LIN {X 0,Y 380.592,Z 511.818,A -85,B 0,C 180,E1 -13079.719,E2 -13079.719} C_VEL
LIN {X 0,Y 375.84,Z 486.306,A -85,B 0,C 180,E1 -13080.73,E2 -13080.73} C_VEL
LIN {X 0,Y 368.954,Z 471.038,A -85,B 0,C 180,E1 -13081.761,E2 -13081.761} C_VEL
LIN {X 0,Y 368.004,Z 468.713,A -85,B 0,C 180,E1 -13081.936,E2 -13081.936} C_VEL
LIN {X 0,Y 364.375,Z 454.654,A -85,B 0,C 180,E1 -13085.353,E2 -13085.353} C_VEL
LIN {X 0,Y 361.868,Z 446.029,A -85,B 0,C 180,E1 -13087.61,E2 -13087.61} C_VEL
LIN {X 0,Y 361.87,Z 446.036,A -85,B 0,C 180,E1 -13091.323,E2 -13091.323} C_VEL
LIN {X 0,Y 361.898,Z 446.033,A -85,B 0,C 180,E1 -13094.354,E2 -13094.354} C_VEL
LIN {X 0,Y 361.831,Z 446.035,A -85,B 0,C 180,E1 -13097.567,E2 -13097.567} C_VEL
LIN {X 0,Y 361.865,Z 446.035,A -85,B 0,C 180,E1 -13100.973,E2 -13100.973} C_VEL
LIN {X 0,Y 361.868,Z 446.032,A -85,B 0,C 180,E1 -13104.655,E2 -13104.655} C_VEL
LIN {X 0,Y 361.831,Z 446.041,A -85,B 0,C 180,E1 -13108.37,E2 -13108.37} C_VEL
LIN {X 0,Y 361.901,Z 446.029,A -85,B 0,C 180,E1 -13112.221,E2 -13112.221} C_VEL
LIN {X 0,Y 361.921,Z 446.028,A -85,B 0,C 180,E1 -13114.71,E2 -13114.71} C_VEL
LIN {X 0,Y 361.885,Z 446.032,A -85,B 0,C 180,E1 -13118.347,E2 -13118.347} C_VEL
LIN {X 0,Y 361.96,Z 446.023,A -85,B 0,C 180,E1 -13122.061,E2 -13122.061} C_VEL
LIN {X 0,Y 361.991,Z 446.016,A -85,B 0,C 180,E1 -13126.101,E2 -13126.101} C_VEL
LIN {X 0,Y 362.029,Z 446.01,A -85,B 0,C 180,E1 -13129.938,E2 -13129.938} C_VEL
LIN {X 0,Y 362.144,Z 446.001,A -85,B 0,C 180,E1 -13132.193,E2 -13132.193} C_VEL
LIN {X 0,Y 362.112,Z 445.999,A -85,B 0,C 180,E1 -13134.431,E2 -13134.431} C_VEL
LIN {X 0,Y 362.276,Z 445.977,A -85,B 0,C 180,E1 -13137.777,E2 -13137.777} C_VEL
LIN {X 0,Y 362.421,Z 445.967,A -85,B 0,C 180,E1 -13140,E2 -13140} C_VEL
LIN {X 0,Y 362.276,Z 445.979,A -85,B 0,C 180,E1 -13142.224,E2 -13142.224} C_VEL
LIN {X 0,Y 362.165,Z 445.997,A -85,B 0,C 180,E1 -13146.687,E2 -13146.687} C_VEL
LIN {X 0,Y 362.067,Z 446.01,A -85,B 0,C 180,E1 -13148.934,E2 -13148.934} C_VEL
LIN {X 0,Y 361.954,Z 446.024,A -85,B 0,C 180,E1 -13152.333,E2 -13152.333} C_VEL
LIN {X 0,Y 361.957,Z 446.022,A -85,B 0,C 180,E1 -13154.621,E2 -13154.621} C_VEL
LIN {X 0,Y 361.954,Z 446.026,A -85,B 0,C 180,E1 -13158.1,E2 -13158.1} C_VEL
LIN {X 0,Y 361.886,Z 446.03,A -85,B 0,C 180,E1 -13161.654,E2 -13161.654} C_VEL
LIN {X 0,Y 361.923,Z 446.03,A -85,B 0,C 180,E1 -13165.291,E2 -13165.291} C_VEL
LIN {X 0,Y 361.917,Z 446.03,A -85,B 0,C 180,E1 -13167.779,E2 -13167.779} C_VEL
LIN {X 0,Y 361.855,Z 446.037,A -85,B 0,C 180,E1 -13171.628,E2 -13171.628} C_VEL
LIN {X 0,Y 361.898,Z 446.125,A -85,B 0,C 180,E1 -13173.963,E2 -13173.963} C_VEL
LIN {X 0,Y 363.631,Z 452.4,A -85,B 0,C 180,E1 -13175.693,E2 -13175.693} C_VEL
LIN {X 0,Y 374.505,Z 473.576,A -85,B 0,C 180,E1 -13177.307,E2 -13177.307} C_VEL
LIN {X 0,Y 381.161,Z 488.749,A -85,B 0,C 180,E1 -13178.277,E2 -13178.277} C_VEL
LIN {X 0,Y 377.634,Z 617.32,A -85,B 0,C 180,E1 -13180.831,E2 -13180.831} C_VEL
LIN {X 0,Y 376.702,Z 633.034,A -85,B 0,C 180,E1 -13181.362,E2 -13181.362} C_VEL
LIN {X 0,Y 375.589,Z 647.26,A -85,B 0,C 180,E1 -13182.05,E2 -13182.05} C_VEL
LIN {X 0,Y 374.132,Z 661.968,A -85,B 0,C 180,E1 -13182.995,E2 -13182.995} C_VEL
LIN {X 0,Y 372.388,Z 676.407,A -85,B 0,C 180,E1 -13184.181,E2 -13184.181} C_VEL
LIN {X 0,Y 370.685,Z 688.967,A -85,B 0,C 180,E1 -13185.454,E2 -13185.454} C_VEL
LIN {X 0,Y 368.931,Z 700.675,A -85,B 0,C 180,E1 -13186.891,E2 -13186.891} C_VEL
LIN {X 0,Y 367.053,Z 712.573,A -85,B 0,C 180,E1 -13188.658,E2 -13188.658} C_VEL
LIN {X 0,Y 365.247,Z 723.245,A -85,B 0,C 180,E1 -13190.583,E2 -13190.583} C_VEL
LIN {X 0,Y 364.044,Z 731.254,A -85,B 0,C 180,E1 -13192.328,E2 -13192.328} C_VEL
LIN {X 0,Y 362.703,Z 739.466,A -85,B 0,C 180,E1 -13194.472,E2 -13194.472} C_VEL
LIN {X 0,Y 361.751,Z 746.21,A -85,B 0,C 180,E1 -13196.657,E2 -13196.657} C_VEL
LIN {X 0,Y 361.075,Z 751.703,A -85,B 0,C 180,E1 -13198.918,E2 -13198.918} C_VEL
LIN {X 0,Y 360.532,Z 756.05,A -85,B 0,C 180,E1 -13201.308,E2 -13201.308} C_VEL
LIN {X 0,Y 360.22,Z 759.126,A -85,B 0,C 180,E1 -13203.829,E2 -13203.829} C_VEL
LIN {X 0,Y 360.067,Z 760.813,A -85,B 0,C 180,E1 -13206.546,E2 -13206.546} C_VEL
LIN {X 0,Y 360.056,Z 760.99,A -85,B 0,C 180,E1 -13208.232,E2 -13208.232} C_VEL
LIN {X 0,Y 360.152,Z 760.166,A -85,B 0,C 180,E1 -13210.627,E2 -13210.627} C_VEL
LIN {X 0,Y 360.35,Z 758.07,A -85,B 0,C 180,E1 -13212.99,E2 -13212.99} C_VEL
LIN {X 0,Y 360.698,Z 754.681,A -85,B 0,C 180,E1 -13215.328,E2 -13215.328} C_VEL
LIN {X 0,Y 361.143,Z 749.972,A -85,B 0,C 180,E1 -13217.64,E2 -13217.64} C_VEL
LIN {X 0,Y 361.874,Z 743.855,A -85,B 0,C 180,E1 -13219.934,E2 -13219.934} C_VEL
LIN {X 0,Y 362.924,Z 736.176,A -85,B 0,C 180,E1 -13222.21,E2 -13222.21} C_VEL
LIN {X 0,Y 364.092,Z 727.96,A -85,B 0,C 180,E1 -13224.184,E2 -13224.184} C_VEL
LIN {X 0,Y 365.644,Z 718.092,A -85,B 0,C 180,E1 -13226.144,E2 -13226.144} C_VEL
LIN {X 0,Y 367.185,Z 708.015,A -85,B 0,C 180,E1 -13227.807,E2 -13227.807} C_VEL
LIN {X 0,Y 368.887,Z 696.077,A -85,B 0,C 180,E1 -13229.455,E2 -13229.455} C_VEL
LIN {X 0,Y 370.57,Z 684.121,A -85,B 0,C 180,E1 -13230.816,E2 -13230.816} C_VEL
LIN {X 0,Y 372.187,Z 671.209,A -85,B 0,C 180,E1 -13232.03,E2 -13232.03} C_VEL
LIN {X 0,Y 373.735,Z 656.677,A -85,B 0,C 180,E1 -13233.128,E2 -13233.128} C_VEL
LIN {X 0,Y 374.985,Z 642.461,A -85,B 0,C 180,E1 -13233.963,E2 -13233.963} C_VEL
LIN {X 0,Y 376.031,Z 627.288,A -85,B 0,C 180,E1 -13234.624,E2 -13234.624} C_VEL
LIN {X 0,Y 376.736,Z 611.413,A -85,B 0,C 180,E1 -13235.084,E2 -13235.084} C_VEL
LIN {X 0,Y 377.665,Z 575.869,A -85,B 0,C 180,E1 -13235.78,E2 -13235.78} C_VEL
LIN {X 0,Y 377.269,Z 570.066,A -85,B 0,C 180,E1 -13235.934,E2 -13235.934} C_VEL
LIN {X 0,Y 372.626,Z 551.43,A -85,B 0,C 180,E1 -13236.7,E2 -13236.7} C_VEL
LIN {X 0,Y 372.167,Z 545.629,A -85,B 0,C 180,E1 -13236.864,E2 -13236.864} C_VEL
LIN {X 0,Y 373.609,Z 489.608,A -85,B 0,C 180,E1 -13237.975,E2 -13237.975} C_VEL
LIN {X 0,Y 364.5,Z 468.659,A -85,B 0,C 180,E1 -13239.245,E2 -13239.245} C_VEL
LIN {X 0,Y 356.131,Z 451.447,A -85,B 0,C 180,E1 -13240.457,E2 -13240.457} C_VEL
LIN {X 0,Y 354.915,Z 446.893,A -85,B 0,C 180,E1 -13241.711,E2 -13241.711} C_VEL
LIN {X 0,Y 354.924,Z 446.901,A -85,B 0,C 180,E1 -13244.917,E2 -13244.917} C_VEL
LIN {X 0,Y 354.913,Z 446.898,A -85,B 0,C 180,E1 -13248.472,E2 -13248.472} C_VEL
LIN {X 0,Y 354.842,Z 446.912,A -85,B 0,C 180,E1 -13252.106,E2 -13252.106} C_VEL
LIN {X 0,Y 354.903,Z 446.904,A -85,B 0,C 180,E1 -13255.827,E2 -13255.827} C_VEL
LIN {X 0,Y 354.858,Z 446.907,A -85,B 0,C 180,E1 -13259.679,E2 -13259.679} C_VEL
LIN {X 0,Y 354.809,Z 446.907,A -85,B 0,C 180,E1 -13263.702,E2 -13263.702} C_VEL
LIN {X 0,Y 354.802,Z 446.91,A -85,B 0,C 180,E1 -13266.459,E2 -13266.459} C_VEL
LIN {X 0,Y 354.827,Z 446.904,A -85,B 0,C 180,E1 -13269.424,E2 -13269.424} C_VEL
LIN {X 0,Y 354.793,Z 446.908,A -85,B 0,C 180,E1 -13272.867,E2 -13272.867} C_VEL
LIN {X 0,Y 354.778,Z 446.916,A -85,B 0,C 180,E1 -13276.105,E2 -13276.105} C_VEL
LIN {X 0,Y 354.826,Z 446.901,A -85,B 0,C 180,E1 -13279.184,E2 -13279.184} C_VEL
LIN {X 0,Y 354.811,Z 446.908,A -85,B 0,C 180,E1 -13282.402,E2 -13282.402} C_VEL
LIN {X 0,Y 354.814,Z 446.902,A -85,B 0,C 180,E1 -13284.941,E2 -13284.941} C_VEL
LIN {X 0,Y 354.797,Z 446.909,A -85,B 0,C 180,E1 -13288.404,E2 -13288.404} C_VEL
LIN {X 0,Y 354.848,Z 446.901,A -85,B 0,C 180,E1 -13291.618,E2 -13291.618} C_VEL
LIN {X 0,Y 354.9,Z 446.899,A -85,B 0,C 180,E1 -13294.172,E2 -13294.172} C_VEL
LIN {X 0,Y 354.828,Z 446.902,A -85,B 0,C 180,E1 -13297.893,E2 -13297.893} C_VEL
LIN {X 0,Y 354.924,Z 446.89,A -85,B 0,C 180,E1 -13301.891,E2 -13301.891} C_VEL
LIN {X 0,Y 354.944,Z 446.897,A -85,B 0,C 180,E1 -13305.981,E2 -13305.981} C_VEL
LIN {X 0,Y 354.979,Z 446.878,A -85,B 0,C 180,E1 -13309.736,E2 -13309.736} C_VEL
LIN {X 0,Y 355.115,Z 446.871,A -85,B 0,C 180,E1 -13312.037,E2 -13312.037} C_VEL
LIN {X 0,Y 355.093,Z 446.875,A -85,B 0,C 180,E1 -13314.32,E2 -13314.32} C_VEL
LIN {X 0,Y 355.244,Z 446.846,A -85,B 0,C 180,E1 -13317.732,E2 -13317.732} C_VEL
LIN {X 0,Y 355.398,Z 446.841,A -85,B 0,C 180,E1 -13320,E2 -13320} C_VEL
LIN {X 0,Y 355.246,Z 446.851,A -85,B 0,C 180,E1 -13322.267,E2 -13322.267} C_VEL
LIN {X 0,Y 355.138,Z 446.865,A -85,B 0,C 180,E1 -13326.819,E2 -13326.819} C_VEL
LIN {X 0,Y 355.015,Z 446.886,A -85,B 0,C 180,E1 -13329.112,E2 -13329.112} C_VEL
LIN {X 0,Y 354.921,Z 446.884,A -85,B 0,C 180,E1 -13332.581,E2 -13332.581} C_VEL
LIN {X 0,Y 354.889,Z 446.901,A -85,B 0,C 180,E1 -13336.096,E2 -13336.096} C_VEL
LIN {X 0,Y 354.901,Z 446.884,A -85,B 0,C 180,E1 -13338.472,E2 -13338.472} C_VEL
LIN {X 0,Y 354.835,Z 446.909,A -85,B 0,C 180,E1 -13342.106,E2 -13342.106} C_VEL
LIN {X 0,Y 354.899,Z 446.901,A -85,B 0,C 180,E1 -13345.827,E2 -13345.827} C_VEL
LIN {X 0,Y 354.854,Z 446.91,A -85,B 0,C 180,E1 -13349.678,E2 -13349.678} C_VEL
LIN {X 0,Y 354.806,Z 446.913,A -85,B 0,C 180,E1 -13353.702,E2 -13353.702} C_VEL
LIN {X 0,Y 354.801,Z 446.913,A -85,B 0,C 180,E1 -13356.459,E2 -13356.459} C_VEL
LIN {X 0,Y 354.824,Z 446.913,A -85,B 0,C 180,E1 -13359.423,E2 -13359.423} C_VEL
LIN {X 0,Y 354.791,Z 446.914,A -85,B 0,C 180,E1 -13362.867,E2 -13362.867} C_VEL
LIN {X 0,Y 354.851,Z 446.907,A -85,B 0,C 180,E1 -13366.116,E2 -13366.116} C_VEL
LIN {X 0,Y 354.856,Z 446.909,A -85,B 0,C 180,E1 -13369.188,E2 -13369.188} C_VEL
LIN {X 0,Y 354.832,Z 446.935,A -85,B 0,C 180,E1 -13372.597,E2 -13372.597} C_VEL
LIN {X 0,Y 358.374,Z 460.009,A -85,B 0,C 180,E1 -13375.824,E2 -13375.824} C_VEL
LIN {X 0,Y 360.621,Z 469.402,A -85,B 0,C 180,E1 -13378.014,E2 -13378.014} C_VEL
LIN {X 0,Y 368.425,Z 487.379,A -85,B 0,C 180,E1 -13379.138,E2 -13379.138} C_VEL
LIN {X 0,Y 373.23,Z 513.749,A -85,B 0,C 180,E1 -13380.135,E2 -13380.135} C_VEL
LIN {X 0,Y 369.957,Z 635.975,A -85,B 0,C 180,E1 -13382.569,E2 -13382.569} C_VEL
LIN {X 0,Y 368.945,Z 652.02,A -85,B 0,C 180,E1 -13383.101,E2 -13383.101} C_VEL
LIN {X 0,Y 367.762,Z 666.067,A -85,B 0,C 180,E1 -13383.773,E2 -13383.773} C_VEL
LIN {X 0,Y 366.127,Z 681.117,A -85,B 0,C 180,E1 -13384.724,E2 -13384.724} C_VEL
LIN {X 0,Y 364.458,Z 694.507,A -85,B 0,C 180,E1 -13385.809,E2 -13385.809} C_VEL
LIN {X 0,Y 362.564,Z 708.251,A -85,B 0,C 180,E1 -13387.189,E2 -13387.189} C_VEL
LIN {X 0,Y 360.698,Z 720.702,A -85,B 0,C 180,E1 -13388.721,E2 -13388.721} C_VEL
LIN {X 0,Y 359.084,Z 731.85,A -85,B 0,C 180,E1 -13390.384,E2 -13390.384} C_VEL
LIN {X 0,Y 357.371,Z 742.327,A -85,B 0,C 180,E1 -13392.252,E2 -13392.252} C_VEL
LIN {X 0,Y 355.992,Z 751.579,A -85,B 0,C 180,E1 -13394.249,E2 -13394.249} C_VEL
LIN {X 0,Y 354.917,Z 759.263,A -85,B 0,C 180,E1 -13396.253,E2 -13396.253} C_VEL
LIN {X 0,Y 354.138,Z 766.441,A -85,B 0,C 180,E1 -13398.553,E2 -13398.553} C_VEL
LIN {X 0,Y 353.593,Z 772.091,A -85,B 0,C 180,E1 -13400.85,E2 -13400.85} C_VEL
LIN {X 0,Y 353.305,Z 776.376,A -85,B 0,C 180,E1 -13403.145,E2 -13403.145} C_VEL
LIN {X 0,Y 353.226,Z 779.396,A -85,B 0,C 180,E1 -13405.435,E2 -13405.435} C_VEL
LIN {X 0,Y 353.161,Z 781.216,A -85,B 0,C 180,E1 -13407.718,E2 -13407.718} C_VEL
LIN {X 0,Y 353.26,Z 781.847,A -85,B 0,C 180,E1 -13409.999,E2 -13409.999} C_VEL
LIN {X 0,Y 353.163,Z 781.288,A -85,B 0,C 180,E1 -13412.28,E2 -13412.28} C_VEL
LIN {X 0,Y 353.23,Z 779.582,A -85,B 0,C 180,E1 -13414.564,E2 -13414.564} C_VEL
LIN {X 0,Y 353.307,Z 776.695,A -85,B 0,C 180,E1 -13416.854,E2 -13416.854} C_VEL
LIN {X 0,Y 353.595,Z 772.565,A -85,B 0,C 180,E1 -13419.148,E2 -13419.148} C_VEL
LIN {X 0,Y 354.147,Z 767.089,A -85,B 0,C 180,E1 -13421.445,E2 -13421.445} C_VEL
LIN {X 0,Y 354.932,Z 760.119,A -85,B 0,C 180,E1 -13423.745,E2 -13423.745} C_VEL
LIN {X 0,Y 356.241,Z 751.456,A -85,B 0,C 180,E1 -13426.032,E2 -13426.032} C_VEL
LIN {X 0,Y 357.654,Z 742.271,A -85,B 0,C 180,E1 -13428.028,E2 -13428.028} C_VEL
LIN {X 0,Y 359.443,Z 732.115,A -85,B 0,C 180,E1 -13429.852,E2 -13429.852} C_VEL
LIN {X 0,Y 361.319,Z 719.822,A -85,B 0,C 180,E1 -13431.688,E2 -13431.688} C_VEL
LIN {X 0,Y 363.338,Z 707.348,A -85,B 0,C 180,E1 -13433.21,E2 -13433.21} C_VEL
LIN {X 0,Y 365.348,Z 693.568,A -85,B 0,C 180,E1 -13434.581,E2 -13434.581} C_VEL
LIN {X 0,Y 367.116,Z 680.319,A -85,B 0,C 180,E1 -13435.646,E2 -13435.646} C_VEL
LIN {X 0,Y 368.663,Z 666.134,A -85,B 0,C 180,E1 -13436.553,E2 -13436.553} C_VEL
LIN {X 0,Y 370.033,Z 651.123,A -85,B 0,C 180,E1 -13437.27,E2 -13437.27} C_VEL
LIN {X 0,Y 371.091,Z 634.97,A -85,B 0,C 180,E1 -13437.798,E2 -13437.798} C_VEL
LIN {X 0,Y 373.955,Z 535.217,A -85,B 0,C 180,E1 -13439.8,E2 -13439.8} C_VEL
LIN {X 0,Y 374.492,Z 513.151,A -85,B 0,C 180,E1 -13440.248,E2 -13440.248} C_VEL
LIN {X 0,Y 370.649,Z 491.854,A -85,B 0,C 180,E1 -13441.105,E2 -13441.105} C_VEL
LIN {X 0,Y 369.765,Z 488.167,A -85,B 0,C 180,E1 -13441.279,E2 -13441.279} C_VEL
LIN {X 0,Y 362.335,Z 471.976,A -85,B 0,C 180,E1 -13442.428,E2 -13442.428} C_VEL
LIN {X 0,Y 360.715,Z 468.458,A -85,B 0,C 180,E1 -13442.71,E2 -13442.71} C_VEL
LIN {X 0,Y 357.939,Z 457.559,A -85,B 0,C 180,E1 -13445.43,E2 -13445.43} C_VEL
LIN {X 0,Y 354.848,Z 446.907,A -85,B 0,C 180,E1 -13448.327,E2 -13448.327} C_VEL
LIN {X 0,Y 354.834,Z 446.913,A -85,B 0,C 180,E1 -13451.18,E2 -13451.18} C_VEL
LIN {X 0,Y 354.85,Z 446.913,A -85,B 0,C 180,E1 -13454.521,E2 -13454.521} C_VEL
LIN {X 0,Y 354.789,Z 446.912,A -85,B 0,C 180,E1 -13457.662,E2 -13457.662} C_VEL
LIN {X 0,Y 354.809,Z 446.916,A -85,B 0,C 180,E1 -13460.665,E2 -13460.665} C_VEL
LIN {X 0,Y 354.816,Z 446.91,A -85,B 0,C 180,E1 -13464.3,E2 -13464.3} C_VEL
LIN {X 0,Y 354.781,Z 446.913,A -85,B 0,C 180,E1 -13467.666,E2 -13467.666} C_VEL
LIN {X 0,Y 354.839,Z 446.909,A -85,B 0,C 180,E1 -13471.618,E2 -13471.618} C_VEL
LIN {X 0,Y 354.892,Z 446.902,A -85,B 0,C 180,E1 -13474.172,E2 -13474.172} C_VEL
LIN {X 0,Y 354.827,Z 446.911,A -85,B 0,C 180,E1 -13477.894,E2 -13477.894} C_VEL
LIN {X 0,Y 354.916,Z 446.901,A -85,B 0,C 180,E1 -13481.891,E2 -13481.891} C_VEL
LIN {X 0,Y 354.936,Z 446.895,A -85,B 0,C 180,E1 -13485.981,E2 -13485.981} C_VEL
LIN {X 0,Y 354.975,Z 446.89,A -85,B 0,C 180,E1 -13489.736,E2 -13489.736} C_VEL
LIN {X 0,Y 355.107,Z 446.876,A -85,B 0,C 180,E1 -13492.037,E2 -13492.037} C_VEL
LIN {X 0,Y 355.086,Z 446.873,A -85,B 0,C 180,E1 -13494.321,E2 -13494.321} C_VEL
LIN {X 0,Y 355.239,Z 446.853,A -85,B 0,C 180,E1 -13497.733,E2 -13497.733} C_VEL
LIN {X 0,Y 355.39,Z 446.842,A -85,B 0,C 180,E1 -13500,E2 -13500} C_VEL
LIN {X 0,Y 355.24,Z 446.856,A -85,B 0,C 180,E1 -13502.268,E2 -13502.268} C_VEL
LIN {X 0,Y 355.131,Z 446.872,A -85,B 0,C 180,E1 -13506.82,E2 -13506.82} C_VEL
LIN {X 0,Y 355.008,Z 446.888,A -85,B 0,C 180,E1 -13509.113,E2 -13509.113} C_VEL
LIN {X 0,Y 354.915,Z 446.902,A -85,B 0,C 180,E1 -13512.581,E2 -13512.581} C_VEL
LIN {X 0,Y 354.885,Z 446.904,A -85,B 0,C 180,E1 -13516.096,E2 -13516.096} C_VEL
LIN {X 0,Y 354.901,Z 446.902,A -85,B 0,C 180,E1 -13518.472,E2 -13518.472} C_VEL
LIN {X 0,Y 354.829,Z 446.912,A -85,B 0,C 180,E1 -13522.107,E2 -13522.107} C_VEL
LIN {X 0,Y 354.894,Z 446.9,A -85,B 0,C 180,E1 -13525.828,E2 -13525.828} C_VEL
LIN {X 0,Y 354.85,Z 446.902,A -85,B 0,C 180,E1 -13529.679,E2 -13529.679} C_VEL
LIN {X 0,Y 354.851,Z 447.029,A -85,B 0,C 180,E1 -13533.298,E2 -13533.298} C_VEL
LIN {X 0,Y 356.508,Z 452.708,A -85,B 0,C 180,E1 -13534.912,E2 -13534.912} C_VEL
LIN {X 0,Y 366.72,Z 472.308,A -85,B 0,C 180,E1 -13536.496,E2 -13536.496} C_VEL
LIN {X 0,Y 373.736,Z 487.682,A -85,B 0,C 180,E1 -13537.557,E2 -13537.557} C_VEL
LIN {X 0,Y 375.084,Z 490.9,A -85,B 0,C 180,E1 -13537.759,E2 -13537.759} C_VEL
LIN {X 0,Y 371.442,Z 617.344,A -85,B 0,C 180,E1 -13540.305,E2 -13540.305} C_VEL
LIN {X 0,Y 370.464,Z 633.236,A -85,B 0,C 180,E1 -13540.848,E2 -13540.848} C_VEL
LIN {X 0,Y 369.264,Z 647.775,A -85,B 0,C 180,E1 -13541.565,E2 -13541.565} C_VEL
LIN {X 0,Y 367.732,Z 662.434,A -85,B 0,C 180,E1 -13542.526,E2 -13542.526} C_VEL
LIN {X 0,Y 365.89,Z 677.007,A -85,B 0,C 180,E1 -13543.748,E2 -13543.748} C_VEL
LIN {X 0,Y 364.139,Z 689.313,A -85,B 0,C 180,E1 -13545.021,E2 -13545.021} C_VEL
LIN {X 0,Y 362.293,Z 700.99,A -85,B 0,C 180,E1 -13546.478,E2 -13546.478} C_VEL
LIN {X 0,Y 360.415,Z 712.402,A -85,B 0,C 180,E1 -13548.197,E2 -13548.197} C_VEL
LIN {X 0,Y 358.592,Z 722.851,A -85,B 0,C 180,E1 -13550.097,E2 -13550.097} C_VEL
LIN {X 0,Y 357.232,Z 731.06,A -85,B 0,C 180,E1 -13551.901,E2 -13551.901} C_VEL
LIN {X 0,Y 355.837,Z 739.308,A -85,B 0,C 180,E1 -13554.075,E2 -13554.075} C_VEL
LIN {X 0,Y 354.83,Z 746.166,A -85,B 0,C 180,E1 -13556.319,E2 -13556.319} C_VEL
LIN {X 0,Y 354.062,Z 751.665,A -85,B 0,C 180,E1 -13558.599,E2 -13558.599} C_VEL
LIN {X 0,Y 353.521,Z 756.039,A -85,B 0,C 180,E1 -13561.013,E2 -13561.013} C_VEL
LIN {X 0,Y 353.159,Z 759.19,A -85,B 0,C 180,E1 -13563.576,E2 -13563.576} C_VEL
LIN {X 0,Y 353.02,Z 760.508,A -85,B 0,C 180,E1 -13565.288,E2 -13565.288} C_VEL
LIN {X 0,Y 352.949,Z 761.224,A -85,B 0,C 180,E1 -13567.771,E2 -13567.771} C_VEL
LIN {X 0,Y 353.044,Z 760.614,A -85,B 0,C 180,E1 -13570.22,E2 -13570.22} C_VEL
LIN {X 0,Y 353.249,Z 758.62,A -85,B 0,C 180,E1 -13572.742,E2 -13572.742} C_VEL
LIN {X 0,Y 353.546,Z 755.563,A -85,B 0,C 180,E1 -13575.024,E2 -13575.024} C_VEL
LIN {X 0,Y 353.996,Z 751.101,A -85,B 0,C 180,E1 -13577.387,E2 -13577.387} C_VEL
LIN {X 0,Y 354.725,Z 745.247,A -85,B 0,C 180,E1 -13579.729,E2 -13579.729} C_VEL
LIN {X 0,Y 355.727,Z 737.867,A -85,B 0,C 180,E1 -13582.051,E2 -13582.051} C_VEL
LIN {X 0,Y 356.932,Z 729.956,A -85,B 0,C 180,E1 -13584.067,E2 -13584.067} C_VEL
LIN {X 0,Y 358.469,Z 720.452,A -85,B 0,C 180,E1 -13586.066,E2 -13586.066} C_VEL
LIN {X 0,Y 360.019,Z 710.788,A -85,B 0,C 180,E1 -13587.763,E2 -13587.763} C_VEL
LIN {X 0,Y 361.76,Z 699.334,A -85,B 0,C 180,E1 -13589.444,E2 -13589.444} C_VEL
LIN {X 0,Y 363.575,Z 686.738,A -85,B 0,C 180,E1 -13590.97,E2 -13590.97} C_VEL
LIN {X 0,Y 365.414,Z 673.224,A -85,B 0,C 180,E1 -13592.301,E2 -13592.301} C_VEL
LIN {X 0,Y 366.851,Z 660.923,A -85,B 0,C 180,E1 -13593.295,E2 -13593.295} C_VEL
LIN {X 0,Y 368.273,Z 646.11,A -85,B 0,C 180,E1 -13594.241,E2 -13594.241} C_VEL
LIN {X 0,Y 369.454,Z 630.519,A -85,B 0,C 180,E1 -13594.98,E2 -13594.98} C_VEL
LIN {X 0,Y 370.287,Z 614.974,A -85,B 0,C 180,E1 -13595.48,E2 -13595.48} C_VEL
LIN {X 0,Y 372.167,Z 545.629,A -85,B 0,C 180,E1 -13596.864,E2 -13596.864} C_VEL
LIN {X 0,Y 371.719,Z 539.832,A -85,B 0,C 180,E1 -13597.027,E2 -13597.027} C_VEL
LIN {X 0,Y 367.186,Z 521.207,A -85,B 0,C 180,E1 -13597.819,E2 -13597.819} C_VEL
LIN {X 0,Y 366.774,Z 515.41,A -85,B 0,C 180,E1 -13597.984,E2 -13597.984} C_VEL
LIN {X 0,Y 367.318,Z 491.528,A -85,B 0,C 180,E1 -13598.475,E2 -13598.475} C_VEL
LIN {X 0,Y 359.767,Z 474.01,A -85,B 0,C 180,E1 -13599.557,E2 -13599.557} C_VEL
LIN {X 0,Y 352.292,Z 458.452,A -85,B 0,C 180,E1 -13600.642,E2 -13600.642} C_VEL
LIN {X 0,Y 348.881,Z 451.635,A -85,B 0,C 180,E1 -13601.175,E2 -13601.175} C_VEL
LIN {X 0,Y 347.891,Z 447.776,A -85,B 0,C 180,E1 -13602.247,E2 -13602.247} C_VEL
LIN {X 0,Y 347.87,Z 447.776,A -85,B 0,C 180,E1 -13605.227,E2 -13605.227} C_VEL
LIN {X 0,Y 347.863,Z 447.778,A -85,B 0,C 180,E1 -13608.86,E2 -13608.86} C_VEL
LIN {X 0,Y 347.78,Z 447.79,A -85,B 0,C 180,E1 -13612.579,E2 -13612.579} C_VEL
LIN {X 0,Y 347.816,Z 447.779,A -85,B 0,C 180,E1 -13615.109,E2 -13615.109} C_VEL
LIN {X 0,Y 347.816,Z 447.777,A -85,B 0,C 180,E1 -13617.694,E2 -13617.694} C_VEL
LIN {X 0,Y 347.768,Z 447.791,A -85,B 0,C 180,E1 -13620.346,E2 -13620.346} C_VEL
LIN {X 0,Y 347.748,Z 447.792,A -85,B 0,C 180,E1 -13624.464,E2 -13624.464} C_VEL
LIN {X 0,Y 347.778,Z 447.775,A -85,B 0,C 180,E1 -13627.989,E2 -13627.989} C_VEL
LIN {X 0,Y 347.759,Z 447.789,A -85,B 0,C 180,E1 -13631.829,E2 -13631.829} C_VEL
LIN {X 0,Y 347.711,Z 447.794,A -85,B 0,C 180,E1 -13635.026,E2 -13635.026} C_VEL
LIN {X 0,Y 347.77,Z 447.778,A -85,B 0,C 180,E1 -13638.394,E2 -13638.394} C_VEL
LIN {X 0,Y 347.778,Z 447.786,A -85,B 0,C 180,E1 -13642.011,E2 -13642.011} C_VEL
LIN {X 0,Y 347.746,Z 447.787,A -85,B 0,C 180,E1 -13645.536,E2 -13645.536} C_VEL
LIN {X 0,Y 347.748,Z 447.787,A -85,B 0,C 180,E1 -13648.3,E2 -13648.3} C_VEL
LIN {X 0,Y 347.78,Z 447.776,A -85,B 0,C 180,E1 -13650.987,E2 -13650.987} C_VEL
LIN {X 0,Y 347.833,Z 447.785,A -85,B 0,C 180,E1 -13653.607,E2 -13653.607} C_VEL
LIN {X 0,Y 347.787,Z 447.771,A -85,B 0,C 180,E1 -13656.161,E2 -13656.161} C_VEL
LIN {X 0,Y 347.813,Z 447.785,A -85,B 0,C 180,E1 -13659.909,E2 -13659.909} C_VEL
LIN {X 0,Y 347.868,Z 447.766,A -85,B 0,C 180,E1 -13662.359,E2 -13662.359} C_VEL
LIN {X 0,Y 347.899,Z 447.774,A -85,B 0,C 180,E1 -13665.971,E2 -13665.971} C_VEL
LIN {X 0,Y 347.929,Z 447.757,A -85,B 0,C 180,E1 -13669.525,E2 -13669.525} C_VEL
LIN {X 0,Y 348.075,Z 447.745,A -85,B 0,C 180,E1 -13671.874,E2 -13671.874} C_VEL
LIN {X 0,Y 348.068,Z 447.751,A -85,B 0,C 180,E1 -13674.205,E2 -13674.205} C_VEL
LIN {X 0,Y 348.206,Z 447.722,A -85,B 0,C 180,E1 -13677.686,E2 -13677.686} C_VEL
LIN {X 0,Y 348.347,Z 447.719,A -85,B 0,C 180,E1 -13680,E2 -13680} C_VEL
LIN {X 0,Y 348.208,Z 447.728,A -85,B 0,C 180,E1 -13682.313,E2 -13682.313} C_VEL
LIN {X 0,Y 348.106,Z 447.742,A -85,B 0,C 180,E1 -13686.957,E2 -13686.957} C_VEL
LIN {X 0,Y 347.968,Z 447.766,A -85,B 0,C 180,E1 -13689.298,E2 -13689.298} C_VEL
LIN {X 0,Y 347.89,Z 447.76,A -85,B 0,C 180,E1 -13692.839,E2 -13692.839} C_VEL
LIN {X 0,Y 347.839,Z 447.777,A -85,B 0,C 180,E1 -13696.431,E2 -13696.431} C_VEL
LIN {X 0,Y 347.851,Z 447.763,A -85,B 0,C 180,E1 -13698.86,E2 -13698.86} C_VEL
LIN {X 0,Y 347.774,Z 447.786,A -85,B 0,C 180,E1 -13702.579,E2 -13702.579} C_VEL
LIN {X 0,Y 347.813,Z 447.784,A -85,B 0,C 180,E1 -13705.108,E2 -13705.108} C_VEL
LIN {X 0,Y 347.812,Z 447.785,A -85,B 0,C 180,E1 -13707.693,E2 -13707.693} C_VEL
LIN {X 0,Y 347.764,Z 447.788,A -85,B 0,C 180,E1 -13710.346,E2 -13710.346} C_VEL
LIN {X 0,Y 347.744,Z 447.792,A -85,B 0,C 180,E1 -13714.464,E2 -13714.464} C_VEL
LIN {X 0,Y 347.777,Z 447.788,A -85,B 0,C 180,E1 -13717.989,E2 -13717.989} C_VEL
LIN {X 0,Y 347.751,Z 447.793,A -85,B 0,C 180,E1 -13721.83,E2 -13721.83} C_VEL
LIN {X 0,Y 347.797,Z 447.786,A -85,B 0,C 180,E1 -13725.011,E2 -13725.011} C_VEL
LIN {X 0,Y 347.784,Z 447.789,A -85,B 0,C 180,E1 -13728.391,E2 -13728.391} C_VEL
LIN {X 0,Y 347.768,Z 447.816,A -85,B 0,C 180,E1 -13732.012,E2 -13732.012} C_VEL
LIN {X 0,Y 350.905,Z 459.331,A -85,B 0,C 180,E1 -13734.942,E2 -13734.942} C_VEL
LIN {X 0,Y 353.409,Z 469.294,A -85,B 0,C 180,E1 -13737.334,E2 -13737.334} C_VEL
LIN {X 0,Y 362.47,Z 489.838,A -85,B 0,C 180,E1 -13738.663,E2 -13738.663} C_VEL
LIN {X 0,Y 366.955,Z 514.883,A -85,B 0,C 180,E1 -13739.629,E2 -13739.629} C_VEL
LIN {X 0,Y 363.578,Z 636.087,A -85,B 0,C 180,E1 -13742.085,E2 -13742.085} C_VEL
LIN {X 0,Y 362.536,Z 652.005,A -85,B 0,C 180,E1 -13742.625,E2 -13742.625} C_VEL
LIN {X 0,Y 361.241,Z 666.626,A -85,B 0,C 180,E1 -13743.34,E2 -13743.34} C_VEL
LIN {X 0,Y 359.485,Z 682.039,A -85,B 0,C 180,E1 -13744.35,E2 -13744.35} C_VEL
LIN {X 0,Y 357.73,Z 695.528,A -85,B 0,C 180,E1 -13745.479,E2 -13745.479} C_VEL
LIN {X 0,Y 355.785,Z 709.026,A -85,B 0,C 180,E1 -13746.883,E2 -13746.883} C_VEL
LIN {X 0,Y 353.854,Z 721.315,A -85,B 0,C 180,E1 -13748.442,E2 -13748.442} C_VEL
LIN {X 0,Y 352.155,Z 732.541,A -85,B 0,C 180,E1 -13750.167,E2 -13750.167} C_VEL
LIN {X 0,Y 350.541,Z 741.983,A -85,B 0,C 180,E1 -13751.895,E2 -13751.895} C_VEL
LIN {X 0,Y 349.098,Z 751.264,A -85,B 0,C 180,E1 -13753.929,E2 -13753.929} C_VEL
LIN {X 0,Y 347.925,Z 758.972,A -85,B 0,C 180,E1 -13755.971,E2 -13755.971} C_VEL
LIN {X 0,Y 347.104,Z 766.172,A -85,B 0,C 180,E1 -13758.318,E2 -13758.318} C_VEL
LIN {X 0,Y 346.528,Z 771.84,A -85,B 0,C 180,E1 -13760.662,E2 -13760.662} C_VEL
LIN {X 0,Y 346.227,Z 776.138,A -85,B 0,C 180,E1 -13763.004,E2 -13763.004} C_VEL
LIN {X 0,Y 346.126,Z 779.17,A -85,B 0,C 180,E1 -13765.341,E2 -13765.341} C_VEL
LIN {X 0,Y 346.072,Z 781.002,A -85,B 0,C 180,E1 -13767.672,E2 -13767.672} C_VEL
LIN {X 0,Y 346.163,Z 781.637,A -85,B 0,C 180,E1 -13769.999,E2 -13769.999} C_VEL
LIN {X 0,Y 346.075,Z 781.087,A -85,B 0,C 180,E1 -13772.327,E2 -13772.327} C_VEL
LIN {X 0,Y 346.13,Z 779.39,A -85,B 0,C 180,E1 -13774.658,E2 -13774.658} C_VEL
LIN {X 0,Y 346.229,Z 776.515,A -85,B 0,C 180,E1 -13776.995,E2 -13776.995} C_VEL
LIN {X 0,Y 346.547,Z 772.399,A -85,B 0,C 180,E1 -13779.336,E2 -13779.336} C_VEL
LIN {X 0,Y 347.147,Z 766.935,A -85,B 0,C 180,E1 -13781.679,E2 -13781.679} C_VEL
LIN {X 0,Y 347.932,Z 759.976,A -85,B 0,C 180,E1 -13784.027,E2 -13784.027} C_VEL
LIN {X 0,Y 349.344,Z 751.33,A -85,B 0,C 180,E1 -13786.358,E2 -13786.358} C_VEL
LIN {X 0,Y 350.867,Z 742.16,A -85,B 0,C 180,E1 -13788.389,E2 -13788.389} C_VEL
LIN {X 0,Y 352.656,Z 732.326,A -85,B 0,C 180,E1 -13790.193,E2 -13790.193} C_VEL
LIN {X 0,Y 354.52,Z 720.791,A -85,B 0,C 180,E1 -13791.973,E2 -13791.973} C_VEL
LIN {X 0,Y 356.605,Z 708.561,A -85,B 0,C 180,E1 -13793.52,E2 -13793.52} C_VEL
LIN {X 0,Y 358.699,Z 695.138,A -85,B 0,C 180,E1 -13794.913,E2 -13794.913} C_VEL
LIN {X 0,Y 360.666,Z 681.011,A -85,B 0,C 180,E1 -13796.09,E2 -13796.09} C_VEL
LIN {X 0,Y 362.296,Z 666.553,A -85,B 0,C 180,E1 -13797.042,E2 -13797.042} C_VEL
LIN {X 0,Y 363.749,Z 651.457,A -85,B 0,C 180,E1 -13797.782,E2 -13797.782} C_VEL
LIN {X 0,Y 364.856,Z 635.682,A -85,B 0,C 180,E1 -13798.315,E2 -13798.315} C_VEL
LIN {X 0,Y 367.871,Z 536.348,A -85,B 0,C 180,E1 -13800.344,E2 -13800.344} C_VEL
LIN {X 0,Y 368.44,Z 514.367,A -85,B 0,C 180,E1 -13800.799,E2 -13800.799} C_VEL
LIN {X 0,Y 364.523,Z 492.407,A -85,B 0,C 180,E1 -13801.709,E2 -13801.709} C_VEL
LIN {X 0,Y 359.033,Z 479.821,A -85,B 0,C 180,E1 -13802.593,E2 -13802.593} C_VEL
LIN {X 0,Y 353.443,Z 468.249,A -85,B 0,C 180,E1 -13803.516,E2 -13803.516} C_VEL
LIN {X 0,Y 350.731,Z 457.884,A -85,B 0,C 180,E1 -13806.2,E2 -13806.2} C_VEL
LIN {X 0,Y 347.786,Z 447.787,A -85,B 0,C 180,E1 -13809.066,E2 -13809.066} C_VEL
LIN {X 0,Y 347.778,Z 447.79,A -85,B 0,C 180,E1 -13811.825,E2 -13811.825} C_VEL
LIN {X 0,Y 347.79,Z 447.791,A -85,B 0,C 180,E1 -13815.011,E2 -13815.011} C_VEL
LIN {X 0,Y 347.745,Z 447.797,A -85,B 0,C 180,E1 -13818.397,E2 -13818.397} C_VEL
LIN {X 0,Y 347.768,Z 447.789,A -85,B 0,C 180,E1 -13822.011,E2 -13822.011} C_VEL
LIN {X 0,Y 347.738,Z 447.794,A -85,B 0,C 180,E1 -13825.536,E2 -13825.536} C_VEL
LIN {X 0,Y 347.738,Z 447.796,A -85,B 0,C 180,E1 -13828.3,E2 -13828.3} C_VEL
LIN {X 0,Y 347.772,Z 447.79,A -85,B 0,C 180,E1 -13830.987,E2 -13830.987} C_VEL
LIN {X 0,Y 347.824,Z 447.779,A -85,B 0,C 180,E1 -13833.607,E2 -13833.607} C_VEL
LIN {X 0,Y 347.781,Z 447.784,A -85,B 0,C 180,E1 -13836.162,E2 -13836.162} C_VEL
LIN {X 0,Y 347.81,Z 447.778,A -85,B 0,C 180,E1 -13839.909,E2 -13839.909} C_VEL
LIN {X 0,Y 347.859,Z 447.775,A -85,B 0,C 180,E1 -13842.359,E2 -13842.359} C_VEL
LIN {X 0,Y 347.89,Z 447.773,A -85,B 0,C 180,E1 -13845.971,E2 -13845.971} C_VEL
LIN {X 0,Y 347.926,Z 447.768,A -85,B 0,C 180,E1 -13849.526,E2 -13849.526} C_VEL
LIN {X 0,Y 348.067,Z 447.752,A -85,B 0,C 180,E1 -13851.875,E2 -13851.875} C_VEL
LIN {X 0,Y 348.061,Z 447.748,A -85,B 0,C 180,E1 -13854.206,E2 -13854.206} C_VEL
LIN {X 0,Y 348.202,Z 447.729,A -85,B 0,C 180,E1 -13857.687,E2 -13857.687} C_VEL
LIN {X 0,Y 348.339,Z 447.721,A -85,B 0,C 180,E1 -13860,E2 -13860} C_VEL
LIN {X 0,Y 348.202,Z 447.733,A -85,B 0,C 180,E1 -13862.314,E2 -13862.314} C_VEL
LIN {X 0,Y 348.1,Z 447.747,A -85,B 0,C 180,E1 -13866.958,E2 -13866.958} C_VEL
LIN {X 0,Y 347.961,Z 447.766,A -85,B 0,C 180,E1 -13869.299,E2 -13869.299} C_VEL
LIN {X 0,Y 347.883,Z 447.776,A -85,B 0,C 180,E1 -13872.84,E2 -13872.84} C_VEL
LIN {X 0,Y 347.835,Z 447.78,A -85,B 0,C 180,E1 -13876.432,E2 -13876.432} C_VEL
LIN {X 0,Y 347.85,Z 447.778,A -85,B 0,C 180,E1 -13878.861,E2 -13878.861} C_VEL
LIN {X 0,Y 347.769,Z 447.796,A -85,B 0,C 180,E1 -13882.58,E2 -13882.58} C_VEL
LIN {X 0,Y 347.807,Z 447.789,A -85,B 0,C 180,E1 -13885.109,E2 -13885.109} C_VEL
LIN {X 0,Y 347.807,Z 447.787,A -85,B 0,C 180,E1 -13887.695,E2 -13887.695} C_VEL
LIN {X 0,Y 347.766,Z 447.785,A -85,B 0,C 180,E1 -13890.347,E2 -13890.347} C_VEL
LIN {X 0,Y 347.798,Z 447.937,A -85,B 0,C 180,E1 -13892.593,E2 -13892.593} C_VEL
LIN {X 0,Y 349.262,Z 452.935,A -85,B 0,C 180,E1 -13894.067,E2 -13894.067} C_VEL
LIN {X 0,Y 359.465,Z 471.995,A -85,B 0,C 180,E1 -13895.719,E2 -13895.719} C_VEL
LIN {X 0,Y 365.989,Z 485.848,A -85,B 0,C 180,E1 -13896.742,E2 -13896.742} C_VEL
LIN {X 0,Y 368.993,Z 492.761,A -85,B 0,C 180,E1 -13897.208,E2 -13897.208} C_VEL
LIN {X 0,Y 365.327,Z 616.721,A -85,B 0,C 180,E1 -13899.746,E2 -13899.746} C_VEL
LIN {X 0,Y 364.288,Z 632.585,A -85,B 0,C 180,E1 -13900.276,E2 -13900.276} C_VEL
LIN {X 0,Y 363.092,Z 646.993,A -85,B 0,C 180,E1 -13900.987,E2 -13900.987} C_VEL
LIN {X 0,Y 361.516,Z 661.906,A -85,B 0,C 180,E1 -13901.963,E2 -13901.963} C_VEL
LIN {X 0,Y 359.697,Z 676.029,A -85,B 0,C 180,E1 -13903.146,E2 -13903.146} C_VEL
LIN {X 0,Y 357.846,Z 688.263,A -85,B 0,C 180,E1 -13904.408,E2 -13904.408} C_VEL
LIN {X 0,Y 355.886,Z 700.107,A -85,B 0,C 180,E1 -13905.886,E2 -13905.886} C_VEL
LIN {X 0,Y 353.83,Z 712.184,A -85,B 0,C 180,E1 -13907.714,E2 -13907.714} C_VEL
LIN {X 0,Y 351.931,Z 722.576,A -85,B 0,C 180,E1 -13909.624,E2 -13909.624} C_VEL
LIN {X 0,Y 350.401,Z 731.276,A -85,B 0,C 180,E1 -13911.556,E2 -13911.556} C_VEL
LIN {X 0,Y 348.958,Z 739.179,A -85,B 0,C 180,E1 -13913.669,E2 -13913.669} C_VEL
LIN {X 0,Y 347.894,Z 746.008,A -85,B 0,C 180,E1 -13915.922,E2 -13915.922} C_VEL
LIN {X 0,Y 347.071,Z 751.628,A -85,B 0,C 180,E1 -13918.264,E2 -13918.264} C_VEL
LIN {X 0,Y 346.504,Z 756.045,A -85,B 0,C 180,E1 -13920.71,E2 -13920.71} C_VEL
LIN {X 0,Y 346.089,Z 759.263,A -85,B 0,C 180,E1 -13923.318,E2 -13923.318} C_VEL
LIN {X 0,Y 345.957,Z 760.407,A -85,B 0,C 180,E1 -13924.749,E2 -13924.749} C_VEL
LIN {X 0,Y 345.855,Z 761.375,A -85,B 0,C 180,E1 -13927.289,E2 -13927.289} C_VEL
LIN {X 0,Y 345.911,Z 761.009,A -85,B 0,C 180,E1 -13929.795,E2 -13929.795} C_VEL
LIN {X 0,Y 346.095,Z 759.36,A -85,B 0,C 180,E1 -13932.267,E2 -13932.267} C_VEL
LIN {X 0,Y 346.404,Z 756.44,A -85,B 0,C 180,E1 -13934.708,E2 -13934.708} C_VEL
LIN {X 0,Y 346.868,Z 752.221,A -85,B 0,C 180,E1 -13937.123,E2 -13937.123} C_VEL
LIN {X 0,Y 347.578,Z 746.63,A -85,B 0,C 180,E1 -13939.516,E2 -13939.516} C_VEL
LIN {X 0,Y 348.576,Z 739.53,A -85,B 0,C 180,E1 -13941.887,E2 -13941.887} C_VEL
LIN {X 0,Y 349.789,Z 731.931,A -85,B 0,C 180,E1 -13943.946,E2 -13943.946} C_VEL
LIN {X 0,Y 351.327,Z 722.779,A -85,B 0,C 180,E1 -13945.986,E2 -13945.986} C_VEL
LIN {X 0,Y 352.87,Z 713.45,A -85,B 0,C 180,E1 -13947.718,E2 -13947.718} C_VEL
LIN {X 0,Y 354.79,Z 701.473,A -85,B 0,C 180,E1 -13949.575,E2 -13949.575} C_VEL
LIN {X 0,Y 356.644,Z 689.26,A -85,B 0,C 180,E1 -13951.13,E2 -13951.13} C_VEL
LIN {X 0,Y 358.524,Z 676.329,A -85,B 0,C 180,E1 -13952.477,E2 -13952.477} C_VEL
LIN {X 0,Y 360.188,Z 662.658,A -85,B 0,C 180,E1 -13953.636,E2 -13953.636} C_VEL
LIN {X 0,Y 361.684,Z 648.266,A -85,B 0,C 180,E1 -13954.598,E2 -13954.598} C_VEL
LIN {X 0,Y 362.862,Z 633.482,A -85,B 0,C 180,E1 -13955.349,E2 -13955.349} C_VEL
LIN {X 0,Y 363.811,Z 618.129,A -85,B 0,C 180,E1 -13955.891,E2 -13955.891} C_VEL
LIN {X 0,Y 364.696,Z 588.065,A -85,B 0,C 180,E1 -13956.536,E2 -13956.536} C_VEL
LIN {X 0,Y 366.774,Z 515.41,A -85,B 0,C 180,E1 -13957.984,E2 -13957.984} C_VEL
LIN {X 0,Y 366.458,Z 509.536,A -85,B 0,C 180,E1 -13958.144,E2 -13958.144} C_VEL
LIN {X 0,Y 365.327,Z 503.837,A -85,B 0,C 180,E1 -13958.371,E2 -13958.371} C_VEL
LIN {X 0,Y 362.894,Z 496.559,A -85,B 0,C 180,E1 -13958.752,E2 -13958.752} C_VEL
LIN {X 0,Y 358.089,Z 486.224,A -85,B 0,C 180,E1 -13959.429,E2 -13959.429} C_VEL
LIN {X 0,Y 349.7,Z 467.812,A -85,B 0,C 180,E1 -13960.672,E2 -13960.672} C_VEL
LIN {X 0,Y 341.696,Z 451.878,A -85,B 0,C 180,E1 -13961.907,E2 -13961.907} C_VEL
LIN {X 0,Y 340.855,Z 448.653,A -85,B 0,C 180,E1 -13962.882,E2 -13962.882} C_VEL
LIN {X 0,Y 340.824,Z 448.652,A -85,B 0,C 180,E1 -13965.55,E2 -13965.55} C_VEL
LIN {X 0,Y 340.843,Z 448.65,A -85,B 0,C 180,E1 -13968.468,E2 -13968.468} C_VEL
LIN {X 0,Y 340.757,Z 448.663,A -85,B 0,C 180,E1 -13971.857,E2 -13971.857} C_VEL
LIN {X 0,Y 340.776,Z 448.661,A -85,B 0,C 180,E1 -13975.664,E2 -13975.664} C_VEL
LIN {X 0,Y 340.746,Z 448.656,A -85,B 0,C 180,E1 -13978.32,E2 -13978.32} C_VEL
LIN {X 0,Y 340.708,Z 448.671,A -85,B 0,C 180,E1 -13981.044,E2 -13981.044} C_VEL
LIN {X 0,Y 340.721,Z 448.67,A -85,B 0,C 180,E1 -13985.279,E2 -13985.279} C_VEL
LIN {X 0,Y 340.714,Z 448.655,A -85,B 0,C 180,E1 -13988.386,E2 -13988.386} C_VEL
LIN {X 0,Y 340.706,Z 448.665,A -85,B 0,C 180,E1 -13992.046,E2 -13992.046} C_VEL
LIN {X 0,Y 340.659,Z 448.674,A -85,B 0,C 180,E1 -13996.226,E2 -13996.226} C_VEL
LIN {X 0,Y 340.712,Z 448.664,A -85,B 0,C 180,E1 -13999.749,E2 -13999.749} C_VEL
LIN {X 0,Y 340.708,Z 448.662,A -85,B 0,C 180,E1 -14003.258,E2 -14003.258} C_VEL
LIN {X 0,Y 340.696,Z 448.671,A -85,B 0,C 180,E1 -14006.153,E2 -14006.153} C_VEL
LIN {X 0,Y 340.743,Z 448.651,A -85,B 0,C 180,E1 -14010.329,E2 -14010.329} C_VEL
LIN {X 0,Y 340.805,Z 448.656,A -85,B 0,C 180,E1 -14013.02,E2 -14013.02} C_VEL
LIN {X 0,Y 340.756,Z 448.652,A -85,B 0,C 180,E1 -14015.638,E2 -14015.638} C_VEL
LIN {X 0,Y 340.741,Z 448.665,A -85,B 0,C 180,E1 -14019.473,E2 -14019.473} C_VEL
LIN {X 0,Y 340.859,Z 448.641,A -85,B 0,C 180,E1 -14021.984,E2 -14021.984} C_VEL
LIN {X 0,Y 340.87,Z 448.646,A -85,B 0,C 180,E1 -14025.705,E2 -14025.705} C_VEL
LIN {X 0,Y 340.872,Z 448.638,A -85,B 0,C 180,E1 -14029.306,E2 -14029.306} C_VEL
LIN {X 0,Y 341.076,Z 448.62,A -85,B 0,C 180,E1 -14032.898,E2 -14032.898} C_VEL
LIN {X 0,Y 341.168,Z 448.598,A -85,B 0,C 180,E1 -14037.638,E2 -14037.638} C_VEL
LIN {X 0,Y 341.297,Z 448.598,A -85,B 0,C 180,E1 -14040,E2 -14040} C_VEL
LIN {X 0,Y 341.17,Z 448.604,A -85,B 0,C 180,E1 -14042.361,E2 -14042.361} C_VEL
LIN {X 0,Y 341.076,Z 448.618,A -85,B 0,C 180,E1 -14047.101,E2 -14047.101} C_VEL
LIN {X 0,Y 340.871,Z 448.639,A -85,B 0,C 180,E1 -14050.693,E2 -14050.693} C_VEL
LIN {X 0,Y 340.863,Z 448.649,A -85,B 0,C 180,E1 -14054.325,E2 -14054.325} C_VEL
LIN {X 0,Y 340.837,Z 448.635,A -85,B 0,C 180,E1 -14058.466,E2 -14058.466} C_VEL
LIN {X 0,Y 340.754,Z 448.665,A -85,B 0,C 180,E1 -14061.857,E2 -14061.857} C_VEL
LIN {X 0,Y 340.773,Z 448.661,A -85,B 0,C 180,E1 -14065.664,E2 -14065.664} C_VEL
LIN {X 0,Y 340.742,Z 448.662,A -85,B 0,C 180,E1 -14068.319,E2 -14068.319} C_VEL
LIN {X 0,Y 340.704,Z 448.667,A -85,B 0,C 180,E1 -14071.044,E2 -14071.044} C_VEL
LIN {X 0,Y 340.719,Z 448.669,A -85,B 0,C 180,E1 -14075.279,E2 -14075.279} C_VEL
LIN {X 0,Y 340.712,Z 448.668,A -85,B 0,C 180,E1 -14078.386,E2 -14078.386} C_VEL
LIN {X 0,Y 340.7,Z 448.67,A -85,B 0,C 180,E1 -14082.045,E2 -14082.045} C_VEL
LIN {X 0,Y 340.737,Z 448.669,A -85,B 0,C 180,E1 -14085.47,E2 -14085.47} C_VEL
LIN {X 0,Y 340.725,Z 448.669,A -85,B 0,C 180,E1 -14088.696,E2 -14088.696} C_VEL
LIN {X 0,Y 340.711,Z 448.68,A -85,B 0,C 180,E1 -14091.396,E2 -14091.396} C_VEL
LIN {X 0,Y 343.843,Z 459.982,A -85,B 0,C 180,E1 -14094.362,E2 -14094.362} C_VEL
LIN {X 0,Y 346.19,Z 469.256,A -85,B 0,C 180,E1 -14096.615,E2 -14096.615} C_VEL
LIN {X 0,Y 355.979,Z 491.042,A -85,B 0,C 180,E1 -14098.096,E2 -14098.096} C_VEL
LIN {X 0,Y 357.116,Z 495.231,A -85,B 0,C 180,E1 -14098.3,E2 -14098.3} C_VEL
LIN {X 0,Y 360.733,Z 515.794,A -85,B 0,C 180,E1 -14099.105,E2 -14099.105} C_VEL
LIN {X 0,Y 357.228,Z 636.16,A -85,B 0,C 180,E1 -14101.584,E2 -14101.584} C_VEL
LIN {X 0,Y 356.166,Z 651.987,A -85,B 0,C 180,E1 -14102.133,E2 -14102.133} C_VEL
LIN {X 0,Y 354.871,Z 665.968,A -85,B 0,C 180,E1 -14102.823,E2 -14102.823} C_VEL
LIN {X 0,Y 353.265,Z 680.048,A -85,B 0,C 180,E1 -14103.741,E2 -14103.741} C_VEL
LIN {X 0,Y 351.208,Z 695.05,A -85,B 0,C 180,E1 -14104.992,E2 -14104.992} C_VEL
LIN {X 0,Y 349.19,Z 708.598,A -85,B 0,C 180,E1 -14106.42,E2 -14106.42} C_VEL
LIN {X 0,Y 347.183,Z 720.925,A -85,B 0,C 180,E1 -14108.007,E2 -14108.007} C_VEL
LIN {X 0,Y 345.368,Z 732.178,A -85,B 0,C 180,E1 -14109.76,E2 -14109.76} C_VEL
LIN {X 0,Y 343.717,Z 741.638,A -85,B 0,C 180,E1 -14111.522,E2 -14111.522} C_VEL
LIN {X 0,Y 342.192,Z 750.944,A -85,B 0,C 180,E1 -14113.596,E2 -14113.596} C_VEL
LIN {X 0,Y 340.95,Z 758.673,A -85,B 0,C 180,E1 -14115.678,E2 -14115.678} C_VEL
LIN {X 0,Y 340.085,Z 765.892,A -85,B 0,C 180,E1 -14118.073,E2 -14118.073} C_VEL
LIN {X 0,Y 339.453,Z 771.577,A -85,B 0,C 180,E1 -14120.466,E2 -14120.466} C_VEL
LIN {X 0,Y 339.146,Z 775.893,A -85,B 0,C 180,E1 -14122.857,E2 -14122.857} C_VEL
LIN {X 0,Y 339.03,Z 778.94,A -85,B 0,C 180,E1 -14125.243,E2 -14125.243} C_VEL
LIN {X 0,Y 338.986,Z 780.785,A -85,B 0,C 180,E1 -14127.623,E2 -14127.623} C_VEL
LIN {X 0,Y 339.066,Z 781.426,A -85,B 0,C 180,E1 -14129.999,E2 -14129.999} C_VEL
LIN {X 0,Y 338.989,Z 780.888,A -85,B 0,C 180,E1 -14132.376,E2 -14132.376} C_VEL
LIN {X 0,Y 339.034,Z 779.203,A -85,B 0,C 180,E1 -14134.756,E2 -14134.756} C_VEL
LIN {X 0,Y 339.147,Z 776.338,A -85,B 0,C 180,E1 -14137.142,E2 -14137.142} C_VEL
LIN {X 0,Y 339.47,Z 772.234,A -85,B 0,C 180,E1 -14139.533,E2 -14139.533} C_VEL
LIN {X 0,Y 340.12,Z 766.78,A -85,B 0,C 180,E1 -14141.924,E2 -14141.924} C_VEL
LIN {X 0,Y 340.998,Z 759.633,A -85,B 0,C 180,E1 -14144.38,E2 -14144.38} C_VEL
LIN {X 0,Y 342.466,Z 751.209,A -85,B 0,C 180,E1 -14146.696,E2 -14146.696} C_VEL
LIN {X 0,Y 344.076,Z 742.065,A -85,B 0,C 180,E1 -14148.765,E2 -14148.765} C_VEL
LIN {X 0,Y 346.074,Z 731.421,A -85,B 0,C 180,E1 -14150.75,E2 -14150.75} C_VEL
LIN {X 0,Y 348.081,Z 719.747,A -85,B 0,C 180,E1 -14152.557,E2 -14152.557} C_VEL
LIN {X 0,Y 350.271,Z 707.358,A -85,B 0,C 180,E1 -14154.129,E2 -14154.129} C_VEL
LIN {X 0,Y 352.466,Z 693.698,A -85,B 0,C 180,E1 -14155.542,E2 -14155.542} C_VEL
LIN {X 0,Y 354.498,Z 679.046,A -85,B 0,C 180,E1 -14156.754,E2 -14156.754} C_VEL
LIN {X 0,Y 356.233,Z 664.328,A -85,B 0,C 180,E1 -14157.7,E2 -14157.7} C_VEL
LIN {X 0,Y 357.765,Z 649.319,A -85,B 0,C 180,E1 -14158.408,E2 -14158.408} C_VEL
LIN {X 0,Y 358.718,Z 635.157,A -85,B 0,C 180,E1 -14158.885,E2 -14158.885} C_VEL
LIN {X 0,Y 361.827,Z 537.513,A -85,B 0,C 180,E1 -14160.912,E2 -14160.912} C_VEL
LIN {X 0,Y 362.436,Z 515.566,A -85,B 0,C 180,E1 -14161.372,E2 -14161.372} C_VEL
LIN {X 0,Y 358.757,Z 494.697,A -85,B 0,C 180,E1 -14162.258,E2 -14162.258} C_VEL
LIN {X 0,Y 351.816,Z 479.44,A -85,B 0,C 180,E1 -14163.408,E2 -14163.408} C_VEL
LIN {X 0,Y 346.178,Z 467.866,A -85,B 0,C 180,E1 -14164.409,E2 -14164.409} C_VEL
LIN {X 0,Y 343.155,Z 456.89,A -85,B 0,C 180,E1 -14167.392,E2 -14167.392} C_VEL
LIN {X 0,Y 340.763,Z 448.656,A -85,B 0,C 180,E1 -14169.807,E2 -14169.807} C_VEL
LIN {X 0,Y 340.733,Z 448.658,A -85,B 0,C 180,E1 -14172.894,E2 -14172.894} C_VEL
LIN {X 0,Y 340.67,Z 448.665,A -85,B 0,C 180,E1 -14176.222,E2 -14176.222} C_VEL
LIN {X 0,Y 340.682,Z 448.672,A -85,B 0,C 180,E1 -14179.752,E2 -14179.752} C_VEL
LIN {X 0,Y 340.699,Z 448.671,A -85,B 0,C 180,E1 -14183.258,E2 -14183.258} C_VEL
LIN {X 0,Y 340.688,Z 448.673,A -85,B 0,C 180,E1 -14186.153,E2 -14186.153} C_VEL
LIN {X 0,Y 340.734,Z 448.663,A -85,B 0,C 180,E1 -14190.329,E2 -14190.329} C_VEL
LIN {X 0,Y 340.796,Z 448.653,A -85,B 0,C 180,E1 -14193.02,E2 -14193.02} C_VEL
LIN {X 0,Y 340.749,Z 448.662,A -85,B 0,C 180,E1 -14195.638,E2 -14195.638} C_VEL
LIN {X 0,Y 340.741,Z 448.659,A -85,B 0,C 180,E1 -14199.474,E2 -14199.474} C_VEL
LIN {X 0,Y 340.851,Z 448.653,A -85,B 0,C 180,E1 -14201.984,E2 -14201.984} C_VEL
LIN {X 0,Y 340.862,Z 448.65,A -85,B 0,C 180,E1 -14205.705,E2 -14205.705} C_VEL
LIN {X 0,Y 340.868,Z 448.647,A -85,B 0,C 180,E1 -14209.306,E2 -14209.306} C_VEL
LIN {X 0,Y 341.069,Z 448.623,A -85,B 0,C 180,E1 -14212.898,E2 -14212.898} C_VEL
LIN {X 0,Y 341.164,Z 448.606,A -85,B 0,C 180,E1 -14217.639,E2 -14217.639} C_VEL
LIN {X 0,Y 341.289,Z 448.599,A -85,B 0,C 180,E1 -14220,E2 -14220} C_VEL
LIN {X 0,Y 341.164,Z 448.61,A -85,B 0,C 180,E1 -14222.362,E2 -14222.362} C_VEL
LIN {X 0,Y 341.069,Z 448.622,A -85,B 0,C 180,E1 -14227.102,E2 -14227.102} C_VEL
LIN {X 0,Y 340.864,Z 448.646,A -85,B 0,C 180,E1 -14230.694,E2 -14230.694} C_VEL
LIN {X 0,Y 340.857,Z 448.648,A -85,B 0,C 180,E1 -14234.325,E2 -14234.325} C_VEL
LIN {X 0,Y 340.832,Z 448.655,A -85,B 0,C 180,E1 -14238.468,E2 -14238.468} C_VEL
LIN {X 0,Y 340.748,Z 448.664,A -85,B 0,C 180,E1 -14241.858,E2 -14241.858} C_VEL
LIN {X 0,Y 340.767,Z 448.66,A -85,B 0,C 180,E1 -14245.665,E2 -14245.665} C_VEL
LIN {X 0,Y 340.738,Z 448.673,A -85,B 0,C 180,E1 -14248.32,E2 -14248.32} C_VEL
LIN {X 0,Y 340.76,Z 448.823,A -85,B 0,C 180,E1 -14251.834,E2 -14251.834} C_VEL
LIN {X 0,Y 341.99,Z 453.128,A -85,B 0,C 180,E1 -14253.168,E2 -14253.168} C_VEL
LIN {X 0,Y 350.978,Z 469.379,A -85,B 0,C 180,E1 -14254.695,E2 -14254.695} C_VEL
LIN {X 0,Y 359.144,Z 485.999,A -85,B 0,C 180,E1 -14256.027,E2 -14256.027} C_VEL
LIN {X 0,Y 363.005,Z 494.908,A -85,B 0,C 180,E1 -14256.65,E2 -14256.65} C_VEL
LIN {X 0,Y 359.169,Z 617.173,A -85,B 0,C 180,E1 -14259.192,E2 -14259.192} C_VEL
LIN {X 0,Y 358.096,Z 632.912,A -85,B 0,C 180,E1 -14259.729,E2 -14259.729} C_VEL
LIN {X 0,Y 356.847,Z 647.344,A -85,B 0,C 180,E1 -14260.453,E2 -14260.453} C_VEL
LIN {X 0,Y 355.176,Z 662.423,A -85,B 0,C 180,E1 -14261.46,E2 -14261.46} C_VEL
LIN {X 0,Y 353.356,Z 676.038,A -85,B 0,C 180,E1 -14262.618,E2 -14262.618} C_VEL
LIN {X 0,Y 351.372,Z 688.683,A -85,B 0,C 180,E1 -14263.942,E2 -14263.942} C_VEL
LIN {X 0,Y 349.341,Z 700.494,A -85,B 0,C 180,E1 -14265.445,E2 -14265.445} C_VEL
LIN {X 0,Y 347.561,Z 710.575,A -85,B 0,C 180,E1 -14266.983,E2 -14266.983} C_VEL
LIN {X 0,Y 345.626,Z 720.635,A -85,B 0,C 180,E1 -14268.796,E2 -14268.796} C_VEL
LIN {X 0,Y 343.723,Z 730.635,A -85,B 0,C 180,E1 -14270.985,E2 -14270.985} C_VEL
LIN {X 0,Y 342.135,Z 739.019,A -85,B 0,C 180,E1 -14273.238,E2 -14273.238} C_VEL
LIN {X 0,Y 340.973,Z 745.92,A -85,B 0,C 180,E1 -14275.535,E2 -14275.535} C_VEL
LIN {X 0,Y 340.129,Z 751.566,A -85,B 0,C 180,E1 -14277.906,E2 -14277.906} C_VEL
LIN {X 0,Y 339.489,Z 756.055,A -85,B 0,C 180,E1 -14280.398,E2 -14280.398} C_VEL
LIN {X 0,Y 339.039,Z 759.333,A -85,B 0,C 180,E1 -14283.045,E2 -14283.045} C_VEL
LIN {X 0,Y 338.82,Z 761.089,A -85,B 0,C 180,E1 -14285.491,E2 -14285.491} C_VEL
LIN {X 0,Y 338.743,Z 761.63,A -85,B 0,C 180,E1 -14288.072,E2 -14288.072} C_VEL
LIN {X 0,Y 338.858,Z 760.857,A -85,B 0,C 180,E1 -14290.62,E2 -14290.62} C_VEL
LIN {X 0,Y 339.086,Z 758.803,A -85,B 0,C 180,E1 -14293.133,E2 -14293.133} C_VEL
LIN {X 0,Y 339.486,Z 755.45,A -85,B 0,C 180,E1 -14295.617,E2 -14295.617} C_VEL
LIN {X 0,Y 340.033,Z 750.789,A -85,B 0,C 180,E1 -14298.073,E2 -14298.073} C_VEL
LIN {X 0,Y 340.859,Z 744.73,A -85,B 0,C 180,E1 -14300.507,E2 -14300.507} C_VEL
LIN {X 0,Y 342.09,Z 737.104,A -85,B 0,C 180,E1 -14302.92,E2 -14302.92} C_VEL
LIN {X 0,Y 343.419,Z 728.948,A -85,B 0,C 180,E1 -14305.011,E2 -14305.011} C_VEL
LIN {X 0,Y 345.13,Z 719.375,A -85,B 0,C 180,E1 -14307.038,E2 -14307.038} C_VEL
LIN {X 0,Y 346.886,Z 709.147,A -85,B 0,C 180,E1 -14308.84,E2 -14308.84} C_VEL
LIN {X 0,Y 348.821,Z 697.285,A -85,B 0,C 180,E1 -14310.578,E2 -14310.578} C_VEL
LIN {X 0,Y 350.684,Z 685.442,A -85,B 0,C 180,E1 -14312.01,E2 -14312.01} C_VEL
LIN {X 0,Y 352.494,Z 672.726,A -85,B 0,C 180,E1 -14313.281,E2 -14313.281} C_VEL
LIN {X 0,Y 354.219,Z 658.717,A -85,B 0,C 180,E1 -14314.41,E2 -14314.41} C_VEL
LIN {X 0,Y 355.621,Z 644.407,A -85,B 0,C 180,E1 -14315.316,E2 -14315.316} C_VEL
LIN {X 0,Y 356.856,Z 628.833,A -85,B 0,C 180,E1 -14316.042,E2 -14316.042} C_VEL
LIN {X 0,Y 357.671,Z 613.489,A -85,B 0,C 180,E1 -14316.523,E2 -14316.523} C_VEL
LIN {X 0,Y 361.126,Z 493.631,A -85,B 0,C 180,E1 -14318.979,E2 -14318.979} C_VEL
LIN {X 0,Y 358.089,Z 486.224,A -85,B 0,C 180,E1 -14319.429,E2 -14319.429} C_VEL
LIN {X 0,Y 355.236,Z 482.374,A -85,B 0,C 180,E1 -14319.787,E2 -14319.787} C_VEL
LIN {X 0,Y 346.374,Z 474.608,A -85,B 0,C 180,E1 -14320.839,E2 -14320.839} C_VEL
LIN {X 0,Y 344.895,Z 472.712,A -85,B 0,C 180,E1 -14321.035,E2 -14321.035} C_VEL
LIN {X 0,Y 335.441,Z 454.296,A -85,B 0,C 180,E1 -14322.502,E2 -14322.502} C_VEL
LIN {X 0,Y 334.505,Z 452.181,A -85,B 0,C 180,E1 -14322.668,E2 -14322.668} C_VEL
LIN {X 0,Y 333.798,Z 449.529,A -85,B 0,C 180,E1 -14323.456,E2 -14323.456} C_VEL
LIN {X 0,Y 333.752,Z 449.539,A -85,B 0,C 180,E1 -14327.146,E2 -14327.146} C_VEL
LIN {X 0,Y 333.751,Z 449.54,A -85,B 0,C 180,E1 -14329.69,E2 -14329.69} C_VEL
LIN {X 0,Y 333.679,Z 449.542,A -85,B 0,C 180,E1 -14333.59,E2 -14333.59} C_VEL
LIN {X 0,Y 333.74,Z 449.538,A -85,B 0,C 180,E1 -14336.246,E2 -14336.246} C_VEL
LIN {X 0,Y 333.715,Z 449.534,A -85,B 0,C 180,E1 -14338.972,E2 -14338.972} C_VEL
LIN {X 0,Y 333.649,Z 449.535,A -85,B 0,C 180,E1 -14342.588,E2 -14342.588} C_VEL
LIN {X 0,Y 333.68,Z 449.542,A -85,B 0,C 180,E1 -14346.139,E2 -14346.139} C_VEL
LIN {X 0,Y 333.653,Z 449.539,A -85,B 0,C 180,E1 -14349.192,E2 -14349.192} C_VEL
LIN {X 0,Y 333.638,Z 449.543,A -85,B 0,C 180,E1 -14352.5,E2 -14352.5} C_VEL
LIN {X 0,Y 333.604,Z 449.555,A -85,B 0,C 180,E1 -14355.956,E2 -14355.956} C_VEL
LIN {X 0,Y 333.659,Z 449.538,A -85,B 0,C 180,E1 -14359.313,E2 -14359.313} C_VEL
LIN {X 0,Y 333.658,Z 449.543,A -85,B 0,C 180,E1 -14362.349,E2 -14362.349} C_VEL
LIN {X 0,Y 333.676,Z 449.537,A -85,B 0,C 180,E1 -14365.341,E2 -14365.341} C_VEL
LIN {X 0,Y 333.692,Z 449.531,A -85,B 0,C 180,E1 -14369.637,E2 -14369.637} C_VEL
LIN {X 0,Y 333.741,Z 449.536,A -85,B 0,C 180,E1 -14372.401,E2 -14372.401} C_VEL
LIN {X 0,Y 333.728,Z 449.536,A -85,B 0,C 180,E1 -14375.09,E2 -14375.09} C_VEL
LIN {X 0,Y 333.677,Z 449.541,A -85,B 0,C 180,E1 -14379.019,E2 -14379.019} C_VEL
LIN {X 0,Y 333.796,Z 449.525,A -85,B 0,C 180,E1 -14381.589,E2 -14381.589} C_VEL
LIN {X 0,Y 333.809,Z 449.524,A -85,B 0,C 180,E1 -14385.576,E2 -14385.576} C_VEL
LIN {X 0,Y 333.835,Z 449.517,A -85,B 0,C 180,E1 -14389.078,E2 -14389.078} C_VEL
LIN {X 0,Y 334.026,Z 449.498,A -85,B 0,C 180,E1 -14392.747,E2 -14392.747} C_VEL
LIN {X 0,Y 333.812,Z 449.527,A -85,B 0,C 180,E1 -14395.169,E2 -14395.169} C_VEL
LIN {X 0,Y 334.106,Z 449.476,A -85,B 0,C 180,E1 -14397.589,E2 -14397.589} C_VEL
LIN {X 0,Y 334.248,Z 449.476,A -85,B 0,C 180,E1 -14400,E2 -14400} C_VEL
LIN {X 0,Y 334.107,Z 449.483,A -85,B 0,C 180,E1 -14402.411,E2 -14402.411} C_VEL
LIN {X 0,Y 334.026,Z 449.497,A -85,B 0,C 180,E1 -14407.252,E2 -14407.252} C_VEL
LIN {X 0,Y 333.834,Z 449.514,A -85,B 0,C 180,E1 -14410.922,E2 -14410.922} C_VEL
LIN {X 0,Y 333.809,Z 449.527,A -85,B 0,C 180,E1 -14414.634,E2 -14414.634} C_VEL
LIN {X 0,Y 333.796,Z 449.512,A -85,B 0,C 180,E1 -14418.654,E2 -14418.654} C_VEL
LIN {X 0,Y 333.693,Z 449.541,A -85,B 0,C 180,E1 -14422.278,E2 -14422.278} C_VEL
LIN {X 0,Y 333.736,Z 449.538,A -85,B 0,C 180,E1 -14426.246,E2 -14426.246} C_VEL
LIN {X 0,Y 333.712,Z 449.538,A -85,B 0,C 180,E1 -14428.972,E2 -14428.972} C_VEL
LIN {X 0,Y 333.646,Z 449.548,A -85,B 0,C 180,E1 -14432.587,E2 -14432.587} C_VEL
LIN {X 0,Y 333.677,Z 449.544,A -85,B 0,C 180,E1 -14436.138,E2 -14436.138} C_VEL
LIN {X 0,Y 333.647,Z 449.549,A -85,B 0,C 180,E1 -14439.192,E2 -14439.192} C_VEL
LIN {X 0,Y 333.634,Z 449.549,A -85,B 0,C 180,E1 -14442.5,E2 -14442.5} C_VEL
LIN {X 0,Y 333.674,Z 449.545,A -85,B 0,C 180,E1 -14445.968,E2 -14445.968} C_VEL
LIN {X 0,Y 333.702,Z 449.543,A -85,B 0,C 180,E1 -14449.304,E2 -14449.304} C_VEL
LIN {X 0,Y 333.676,Z 449.576,A -85,B 0,C 180,E1 -14450.763,E2 -14450.763} C_VEL
LIN {X 0,Y 337.009,Z 461.544,A -85,B 0,C 180,E1 -14453.993,E2 -14453.993} C_VEL
LIN {X 0,Y 338.837,Z 468.762,A -85,B 0,C 180,E1 -14455.838,E2 -14455.838} C_VEL
LIN {X 0,Y 349.09,Z 491.333,A -85,B 0,C 180,E1 -14457.443,E2 -14457.443} C_VEL
LIN {X 0,Y 350.798,Z 495.765,A -85,B 0,C 180,E1 -14457.716,E2 -14457.716} C_VEL
LIN {X 0,Y 354.507,Z 517.033,A -85,B 0,C 180,E1 -14458.571,E2 -14458.571} C_VEL
LIN {X 0,Y 351.308,Z 623.674,A -85,B 0,C 180,E1 -14460.774,E2 -14460.774} C_VEL
LIN {X 0,Y 350.64,Z 640.583,A -85,B 0,C 180,E1 -14461.205,E2 -14461.205} C_VEL
LIN {X 0,Y 349.503,Z 654.886,A -85,B 0,C 180,E1 -14461.759,E2 -14461.759} C_VEL
LIN {X 0,Y 347.979,Z 669.888,A -85,B 0,C 180,E1 -14462.571,E2 -14462.571} C_VEL
LIN {X 0,Y 346.158,Z 684.683,A -85,B 0,C 180,E1 -14463.632,E2 -14463.632} C_VEL
LIN {X 0,Y 344.083,Z 698.84,A -85,B 0,C 180,E1 -14464.923,E2 -14464.923} C_VEL
LIN {X 0,Y 342.037,Z 711.694,A -85,B 0,C 180,E1 -14466.379,E2 -14466.379} C_VEL
LIN {X 0,Y 340.178,Z 722.491,A -85,B 0,C 180,E1 -14467.849,E2 -14467.849} C_VEL
LIN {X 0,Y 338.596,Z 731.807,A -85,B 0,C 180,E1 -14469.337,E2 -14469.337} C_VEL
LIN {X 0,Y 336.928,Z 741.294,A -85,B 0,C 180,E1 -14471.136,E2 -14471.136} C_VEL
LIN {X 0,Y 335.312,Z 750.624,A -85,B 0,C 180,E1 -14473.25,E2 -14473.25} C_VEL
LIN {X 0,Y 333.99,Z 758.644,A -85,B 0,C 180,E1 -14475.455,E2 -14475.455} C_VEL
LIN {X 0,Y 333.078,Z 765.613,A -85,B 0,C 180,E1 -14477.818,E2 -14477.818} C_VEL
LIN {X 0,Y 332.398,Z 771.315,A -85,B 0,C 180,E1 -14480.261,E2 -14480.261} C_VEL
LIN {X 0,Y 332.056,Z 775.647,A -85,B 0,C 180,E1 -14482.704,E2 -14482.704} C_VEL
LIN {X 0,Y 331.939,Z 778.709,A -85,B 0,C 180,E1 -14485.141,E2 -14485.141} C_VEL
LIN {X 0,Y 331.904,Z 780.568,A -85,B 0,C 180,E1 -14487.572,E2 -14487.572} C_VEL
LIN {X 0,Y 331.968,Z 781.215,A -85,B 0,C 180,E1 -14489.999,E2 -14489.999} C_VEL
LIN {X 0,Y 331.906,Z 780.689,A -85,B 0,C 180,E1 -14492.426,E2 -14492.426} C_VEL
LIN {X 0,Y 331.942,Z 779.015,A -85,B 0,C 180,E1 -14494.857,E2 -14494.857} C_VEL
LIN {X 0,Y 332.072,Z 776.162,A -85,B 0,C 180,E1 -14497.295,E2 -14497.295} C_VEL
LIN {X 0,Y 332.41,Z 772.069,A -85,B 0,C 180,E1 -14499.737,E2 -14499.737} C_VEL
LIN {X 0,Y 333.11,Z 766.629,A -85,B 0,C 180,E1 -14502.179,E2 -14502.179} C_VEL
LIN {X 0,Y 334.026,Z 759.703,A -85,B 0,C 180,E1 -14504.624,E2 -14504.624} C_VEL
LIN {X 0,Y 335.588,Z 751.108,A -85,B 0,C 180,E1 -14507.048,E2 -14507.048} C_VEL
LIN {X 0,Y 337.325,Z 741.981,A -85,B 0,C 180,E1 -14509.155,E2 -14509.155} C_VEL
LIN {X 0,Y 339.264,Z 731.957,A -85,B 0,C 180,E1 -14511.073,E2 -14511.073} C_VEL
LIN {X 0,Y 341.108,Z 721.69,A -85,B 0,C 180,E1 -14512.724,E2 -14512.724} C_VEL
LIN {X 0,Y 343.366,Z 709.724,A -85,B 0,C 180,E1 -14514.324,E2 -14514.324} C_VEL
LIN {X 0,Y 345.584,Z 696.654,A -85,B 0,C 180,E1 -14515.765,E2 -14515.765} C_VEL
LIN {X 0,Y 347.752,Z 682.73,A -85,B 0,C 180,E1 -14516.999,E2 -14516.999} C_VEL
LIN {X 0,Y 349.454,Z 669.24,A -85,B 0,C 180,E1 -14517.958,E2 -14517.958} C_VEL
LIN {X 0,Y 351.037,Z 654.503,A -85,B 0,C 180,E1 -14518.758,E2 -14518.758} C_VEL
LIN {X 0,Y 352.331,Z 639.338,A -85,B 0,C 180,E1 -14519.336,E2 -14519.336} C_VEL
LIN {X 0,Y 353.16,Z 620.657,A -85,B 0,C 180,E1 -14519.793,E2 -14519.793} C_VEL
LIN {X 0,Y 356.515,Z 517.858,A -85,B 0,C 180,E1 -14521.933,E2 -14521.933} C_VEL
LIN {X 0,Y 354.003,Z 502.107,A -85,B 0,C 180,E1 -14522.593,E2 -14522.593} C_VEL
LIN {X 0,Y 352.898,Z 497.057,A -85,B 0,C 180,E1 -14522.842,E2 -14522.842} C_VEL
LIN {X 0,Y 346.221,Z 482.302,A -85,B 0,C 180,E1 -14523.992,E2 -14523.992} C_VEL
LIN {X 0,Y 338.9,Z 467.577,A -85,B 0,C 180,E1 -14525.333,E2 -14525.333} C_VEL
LIN {X 0,Y 335.964,Z 457.007,A -85,B 0,C 180,E1 -14528.331,E2 -14528.331} C_VEL
LIN {X 0,Y 333.692,Z 449.539,A -85,B 0,C 180,E1 -14530.636,E2 -14530.636} C_VEL
LIN {X 0,Y 333.673,Z 449.547,A -85,B 0,C 180,E1 -14534.265,E2 -14534.265} C_VEL
LIN {X 0,Y 333.637,Z 449.545,A -85,B 0,C 180,E1 -14537.618,E2 -14537.618} C_VEL
LIN {X 0,Y 333.647,Z 449.55,A -85,B 0,C 180,E1 -14541.201,E2 -14541.201} C_VEL
LIN {X 0,Y 333.67,Z 449.546,A -85,B 0,C 180,E1 -14543.861,E2 -14543.861} C_VEL
LIN {X 0,Y 333.639,Z 449.546,A -85,B 0,C 180,E1 -14547.412,E2 -14547.412} C_VEL
LIN {X 0,Y 333.683,Z 449.545,A -85,B 0,C 180,E1 -14551.026,E2 -14551.026} C_VEL
LIN {X 0,Y 333.728,Z 449.535,A -85,B 0,C 180,E1 -14553.753,E2 -14553.753} C_VEL
LIN {X 0,Y 333.713,Z 449.542,A -85,B 0,C 180,E1 -14557.914,E2 -14557.914} C_VEL
LIN {X 0,Y 333.787,Z 449.532,A -85,B 0,C 180,E1 -14561.589,E2 -14561.589} C_VEL
LIN {X 0,Y 333.801,Z 449.529,A -85,B 0,C 180,E1 -14565.577,E2 -14565.577} C_VEL
LIN {X 0,Y 333.83,Z 449.525,A -85,B 0,C 180,E1 -14569.078,E2 -14569.078} C_VEL
LIN {X 0,Y 334.018,Z 449.502,A -85,B 0,C 180,E1 -14572.748,E2 -14572.748} C_VEL
LIN {X 0,Y 333.807,Z 449.528,A -85,B 0,C 180,E1 -14575.169,E2 -14575.169} C_VEL
LIN {X 0,Y 334.101,Z 449.486,A -85,B 0,C 180,E1 -14577.589,E2 -14577.589} C_VEL
LIN {X 0,Y 334.24,Z 449.477,A -85,B 0,C 180,E1 -14580,E2 -14580} C_VEL
LIN {X 0,Y 334.101,Z 449.49,A -85,B 0,C 180,E1 -14582.412,E2 -14582.412} C_VEL
LIN {X 0,Y 334.019,Z 449.5,A -85,B 0,C 180,E1 -14587.253,E2 -14587.253} C_VEL
LIN {X 0,Y 333.827,Z 449.521,A -85,B 0,C 180,E1 -14590.922,E2 -14590.922} C_VEL
LIN {X 0,Y 333.802,Z 449.528,A -85,B 0,C 180,E1 -14594.635,E2 -14594.635} C_VEL
LIN {X 0,Y 333.791,Z 449.53,A -85,B 0,C 180,E1 -14598.656,E2 -14598.656} C_VEL
LIN {X 0,Y 333.687,Z 449.548,A -85,B 0,C 180,E1 -14602.279,E2 -14602.279} C_VEL
LIN {X 0,Y 333.731,Z 449.532,A -85,B 0,C 180,E1 -14606.247,E2 -14606.247} C_VEL
LIN {X 0,Y 333.707,Z 449.541,A -85,B 0,C 180,E1 -14608.973,E2 -14608.973} C_VEL
LIN {X 0,Y 333.667,Z 449.548,A -85,B 0,C 180,E1 -14610.98,E2 -14610.98} C_VEL
LIN {X 0,Y 334.872,Z 453.603,A -85,B 0,C 180,E1 -14612.239,E2 -14612.239} C_VEL
LIN {X 0,Y 343.888,Z 469.432,A -85,B 0,C 180,E1 -14613.842,E2 -14613.842} C_VEL
LIN {X 0,Y 353.245,Z 488.203,A -85,B 0,C 180,E1 -14615.431,E2 -14615.431} C_VEL
LIN {X 0,Y 357.022,Z 496.918,A -85,B 0,C 180,E1 -14616.066,E2 -14616.066} C_VEL
LIN {X 0,Y 353.101,Z 617.121,A -85,B 0,C 180,E1 -14618.604,E2 -14618.604} C_VEL
LIN {X 0,Y 351.985,Z 632.902,A -85,B 0,C 180,E1 -14619.144,E2 -14619.144} C_VEL
LIN {X 0,Y 350.651,Z 647.671,A -85,B 0,C 180,E1 -14619.894,E2 -14619.894} C_VEL
LIN {X 0,Y 348.868,Z 662.992,A -85,B 0,C 180,E1 -14620.938,E2 -14620.938} C_VEL
LIN {X 0,Y 346.887,Z 677.119,A -85,B 0,C 180,E1 -14622.174,E2 -14622.174} C_VEL
LIN {X 0,Y 344.84,Z 689.67,A -85,B 0,C 180,E1 -14623.525,E2 -14623.525} C_VEL
LIN {X 0,Y 342.578,Z 702.085,A -85,B 0,C 180,E1 -14625.156,E2 -14625.156} C_VEL
LIN {X 0,Y 340.355,Z 713.857,A -85,B 0,C 180,E1 -14627.047,E2 -14627.047} C_VEL
LIN {X 0,Y 338.205,Z 724.442,A -85,B 0,C 180,E1 -14629.114,E2 -14629.114} C_VEL
LIN {X 0,Y 336.5,Z 733.25,A -85,B 0,C 180,E1 -14631.204,E2 -14631.204} C_VEL
LIN {X 0,Y 334.997,Z 740.831,A -85,B 0,C 180,E1 -14633.385,E2 -14633.385} C_VEL
LIN {X 0,Y 333.968,Z 746.489,A -85,B 0,C 180,E1 -14635.377,E2 -14635.377} C_VEL
LIN {X 0,Y 333.14,Z 751.551,A -85,B 0,C 180,E1 -14637.55,E2 -14637.55} C_VEL
LIN {X 0,Y 332.481,Z 756.069,A -85,B 0,C 180,E1 -14640.074,E2 -14640.074} C_VEL
LIN {X 0,Y 331.956,Z 759.418,A -85,B 0,C 180,E1 -14642.774,E2 -14642.774} C_VEL
LIN {X 0,Y 331.722,Z 761.387,A -85,B 0,C 180,E1 -14645.647,E2 -14645.647} C_VEL
LIN {X 0,Y 331.65,Z 761.837,A -85,B 0,C 180,E1 -14647.578,E2 -14647.578} C_VEL
LIN {X 0,Y 331.734,Z 761.276,A -85,B 0,C 180,E1 -14650.187,E2 -14650.187} C_VEL
LIN {X 0,Y 331.975,Z 759.434,A -85,B 0,C 180,E1 -14652.76,E2 -14652.76} C_VEL
LIN {X 0,Y 332.33,Z 756.322,A -85,B 0,C 180,E1 -14655.3,E2 -14655.3} C_VEL
LIN {X 0,Y 332.875,Z 751.907,A -85,B 0,C 180,E1 -14657.812,E2 -14657.812} C_VEL
LIN {X 0,Y 333.713,Z 746.106,A -85,B 0,C 180,E1 -14660.301,E2 -14660.301} C_VEL
LIN {X 0,Y 334.889,Z 738.775,A -85,B 0,C 180,E1 -14662.767,E2 -14662.767} C_VEL
LIN {X 0,Y 336.211,Z 730.936,A -85,B 0,C 180,E1 -14664.904,E2 -14664.904} C_VEL
LIN {X 0,Y 338.063,Z 721.06,A -85,B 0,C 180,E1 -14667.105,E2 -14667.105} C_VEL
LIN {X 0,Y 340.052,Z 710.094,A -85,B 0,C 180,E1 -14669.113,E2 -14669.113} C_VEL
LIN {X 0,Y 342.058,Z 698.362,A -85,B 0,C 180,E1 -14670.884,E2 -14670.884} C_VEL
LIN {X 0,Y 344.137,Z 685.69,A -85,B 0,C 180,E1 -14672.454,E2 -14672.454} C_VEL
LIN {X 0,Y 346.062,Z 672.555,A -85,B 0,C 180,E1 -14673.785,E2 -14673.785} C_VEL
LIN {X 0,Y 347.809,Z 658.552,A -85,B 0,C 180,E1 -14674.927,E2 -14674.927} C_VEL
LIN {X 0,Y 349.289,Z 644.102,A -85,B 0,C 180,E1 -14675.847,E2 -14675.847} C_VEL
LIN {X 0,Y 350.535,Z 628.374,A -85,B 0,C 180,E1 -14676.584,E2 -14676.584} C_VEL
LIN {X 0,Y 351.401,Z 612.57,A -85,B 0,C 180,E1 -14677.073,E2 -14677.073} C_VEL
LIN {X 0,Y 354.983,Z 495.709,A -85,B 0,C 180,E1 -14679.495,E2 -14679.495} C_VEL
LIN {X 0,Y 348.259,Z 479.941,A -85,B 0,C 180,E1 -14680.521,E2 -14680.521} C_VEL
LIN {X 0,Y 344.895,Z 472.712,A -85,B 0,C 180,E1 -14681.035,E2 -14681.035} C_VEL
LIN {X 0,Y 341.776,Z 469.187,A -85,B 0,C 180,E1 -14681.444,E2 -14681.444} C_VEL
LIN {X 0,Y 332.819,Z 461.905,A -85,B 0,C 180,E1 -14682.596,E2 -14682.596} C_VEL
LIN {X 0,Y 331.305,Z 460.099,A -85,B 0,C 180,E1 -14682.812,E2 -14682.812} C_VEL
LIN {X 0,Y 327.287,Z 452.341,A -85,B 0,C 180,E1 -14683.506,E2 -14683.506} C_VEL
LIN {X 0,Y 326.777,Z 450.405,A -85,B 0,C 180,E1 -14684.126,E2 -14684.126} C_VEL
LIN {X 0,Y 326.704,Z 450.413,A -85,B 0,C 180,E1 -14687.528,E2 -14687.528} C_VEL
LIN {X 0,Y 326.677,Z 450.417,A -85,B 0,C 180,E1 -14690.135,E2 -14690.135} C_VEL
LIN {X 0,Y 326.656,Z 450.412,A -85,B 0,C 180,E1 -14694.129,E2 -14694.129} C_VEL
LIN {X 0,Y 326.689,Z 450.416,A -85,B 0,C 180,E1 -14696.858,E2 -14696.858} C_VEL
LIN {X 0,Y 326.643,Z 450.422,A -85,B 0,C 180,E1 -14700.611,E2 -14700.611} C_VEL
LIN {X 0,Y 326.611,Z 450.422,A -85,B 0,C 180,E1 -14704.019,E2 -14704.019} C_VEL
LIN {X 0,Y 326.631,Z 450.412,A -85,B 0,C 180,E1 -14707.239,E2 -14707.239} C_VEL
LIN {X 0,Y 326.585,Z 450.429,A -85,B 0,C 180,E1 -14711.132,E2 -14711.132} C_VEL
LIN {X 0,Y 326.532,Z 450.432,A -85,B 0,C 180,E1 -14714.743,E2 -14714.743} C_VEL
LIN {X 0,Y 326.592,Z 450.415,A -85,B 0,C 180,E1 -14718.156,E2 -14718.156} C_VEL
LIN {X 0,Y 326.645,Z 450.423,A -85,B 0,C 180,E1 -14721.394,E2 -14721.394} C_VEL
LIN {X 0,Y 326.622,Z 450.413,A -85,B 0,C 180,E1 -14724.851,E2 -14724.851} C_VEL
LIN {X 0,Y 326.612,Z 450.428,A -85,B 0,C 180,E1 -14727.456,E2 -14727.456} C_VEL
LIN {X 0,Y 326.649,Z 450.406,A -85,B 0,C 180,E1 -14730.339,E2 -14730.339} C_VEL
LIN {X 0,Y 326.691,Z 450.411,A -85,B 0,C 180,E1 -14734.516,E2 -14734.516} C_VEL
LIN {X 0,Y 326.623,Z 450.419,A -85,B 0,C 180,E1 -14738.543,E2 -14738.543} C_VEL
LIN {X 0,Y 326.746,Z 450.408,A -85,B 0,C 180,E1 -14741.177,E2 -14741.177} C_VEL
LIN {X 0,Y 326.764,Z 450.4,A -85,B 0,C 180,E1 -14745.433,E2 -14745.433} C_VEL
LIN {X 0,Y 326.771,Z 450.398,A -85,B 0,C 180,E1 -14748.839,E2 -14748.839} C_VEL
LIN {X 0,Y 326.98,Z 450.376,A -85,B 0,C 180,E1 -14752.59,E2 -14752.59} C_VEL
LIN {X 0,Y 326.779,Z 450.402,A -85,B 0,C 180,E1 -14755.065,E2 -14755.065} C_VEL
LIN {X 0,Y 327.046,Z 450.355,A -85,B 0,C 180,E1 -14757.536,E2 -14757.536} C_VEL
LIN {X 0,Y 327.199,Z 450.354,A -85,B 0,C 180,E1 -14760,E2 -14760} C_VEL
LIN {X 0,Y 327.048,Z 450.363,A -85,B 0,C 180,E1 -14762.463,E2 -14762.463} C_VEL
LIN {X 0,Y 326.996,Z 450.365,A -85,B 0,C 180,E1 -14766.169,E2 -14766.169} C_VEL
LIN {X 0,Y 326.915,Z 450.386,A -85,B 0,C 180,E1 -14768.655,E2 -14768.655} C_VEL
LIN {X 0,Y 326.734,Z 450.391,A -85,B 0,C 180,E1 -14772.421,E2 -14772.421} C_VEL
LIN {X 0,Y 326.755,Z 450.406,A -85,B 0,C 180,E1 -14774.957,E2 -14774.957} C_VEL
LIN {X 0,Y 326.733,Z 450.392,A -85,B 0,C 180,E1 -14778.838,E2 -14778.838} C_VEL
LIN {X 0,Y 326.621,Z 450.421,A -85,B 0,C 180,E1 -14782.787,E2 -14782.787} C_VEL
LIN {X 0,Y 326.69,Z 450.415,A -85,B 0,C 180,E1 -14785.483,E2 -14785.483} C_VEL
LIN {X 0,Y 326.661,Z 450.421,A -85,B 0,C 180,E1 -14789.659,E2 -14789.659} C_VEL
LIN {X 0,Y 326.608,Z 450.426,A -85,B 0,C 180,E1 -14794.019,E2 -14794.019} C_VEL
LIN {X 0,Y 326.629,Z 450.424,A -85,B 0,C 180,E1 -14797.239,E2 -14797.239} C_VEL
LIN {X 0,Y 326.578,Z 450.43,A -85,B 0,C 180,E1 -14801.131,E2 -14801.131} C_VEL
LIN {X 0,Y 326.586,Z 450.428,A -85,B 0,C 180,E1 -14804.753,E2 -14804.753} C_VEL
LIN {X 0,Y 326.622,Z 450.424,A -85,B 0,C 180,E1 -14808.161,E2 -14808.161} C_VEL
LIN {X 0,Y 326.69,Z 450.566,A -85,B 0,C 180,E1 -14810.137,E2 -14810.137} C_VEL
LIN {X 0,Y 329.971,Z 462.272,A -85,B 0,C 180,E1 -14813.39,E2 -14813.39} C_VEL
LIN {X 0,Y 331.549,Z 468.562,A -85,B 0,C 180,E1 -14815.04,E2 -14815.04} C_VEL
LIN {X 0,Y 342.327,Z 491.92,A -85,B 0,C 180,E1 -14816.783,E2 -14816.783} C_VEL
LIN {X 0,Y 345.038,Z 498.739,A -85,B 0,C 180,E1 -14817.223,E2 -14817.223} C_VEL
LIN {X 0,Y 348.341,Z 517.741,A -85,B 0,C 180,E1 -14818.008,E2 -14818.008} C_VEL
LIN {X 0,Y 344.676,Z 634.67,A -85,B 0,C 180,E1 -14820.491,E2 -14820.491} C_VEL
LIN {X 0,Y 343.488,Z 650.924,A -85,B 0,C 180,E1 -14821.051,E2 -14821.051} C_VEL
LIN {X 0,Y 342.058,Z 665.654,A -85,B 0,C 180,E1 -14821.799,E2 -14821.799} C_VEL
LIN {X 0,Y 340.229,Z 680.754,A -85,B 0,C 180,E1 -14822.826,E2 -14822.826} C_VEL
LIN {X 0,Y 338.319,Z 693.962,A -85,B 0,C 180,E1 -14823.97,E2 -14823.97} C_VEL
LIN {X 0,Y 336.342,Z 706.372,A -85,B 0,C 180,E1 -14825.297,E2 -14825.297} C_VEL
LIN {X 0,Y 334.028,Z 719.007,A -85,B 0,C 180,E1 -14826.928,E2 -14826.928} C_VEL
LIN {X 0,Y 332.095,Z 729.745,A -85,B 0,C 180,E1 -14828.615,E2 -14828.615} C_VEL
LIN {X 0,Y 330.455,Z 739.42,A -85,B 0,C 180,E1 -14830.429,E2 -14830.429} C_VEL
LIN {X 0,Y 328.633,Z 749.037,A -85,B 0,C 180,E1 -14832.578,E2 -14832.578} C_VEL
LIN {X 0,Y 327.293,Z 757.047,A -85,B 0,C 180,E1 -14834.749,E2 -14834.749} C_VEL
LIN {X 0,Y 326.274,Z 763.695,A -85,B 0,C 180,E1 -14836.928,E2 -14836.928} C_VEL
LIN {X 0,Y 325.475,Z 769.792,A -85,B 0,C 180,E1 -14839.423,E2 -14839.423} C_VEL
LIN {X 0,Y 325.063,Z 774.471,A -85,B 0,C 180,E1 -14841.921,E2 -14841.921} C_VEL
LIN {X 0,Y 324.928,Z 777.624,A -85,B 0,C 180,E1 -14844.24,E2 -14844.24} C_VEL
LIN {X 0,Y 324.852,Z 779.563,A -85,B 0,C 180,E1 -14846.278,E2 -14846.278} C_VEL
LIN {X 0,Y 324.828,Z 780.827,A -85,B 0,C 180,E1 -14848.76,E2 -14848.76} C_VEL
LIN {X 0,Y 324.828,Z 780.89,A -85,B 0,C 180,E1 -14851.239,E2 -14851.239} C_VEL
LIN {X 0,Y 324.856,Z 779.805,A -85,B 0,C 180,E1 -14853.721,E2 -14853.721} C_VEL
LIN {X 0,Y 324.946,Z 777.561,A -85,B 0,C 180,E1 -14856.207,E2 -14856.207} C_VEL
LIN {X 0,Y 325.16,Z 774.114,A -85,B 0,C 180,E1 -14858.701,E2 -14858.701} C_VEL
LIN {X 0,Y 325.646,Z 769.379,A -85,B 0,C 180,E1 -14861.199,E2 -14861.199} C_VEL
LIN {X 0,Y 326.548,Z 763.225,A -85,B 0,C 180,E1 -14863.694,E2 -14863.694} C_VEL
LIN {X 0,Y 327.901,Z 755.517,A -85,B 0,C 180,E1 -14866.178,E2 -14866.178} C_VEL
LIN {X 0,Y 329.473,Z 747.282,A -85,B 0,C 180,E1 -14868.338,E2 -14868.338} C_VEL
LIN {X 0,Y 331.548,Z 737.426,A -85,B 0,C 180,E1 -14870.472,E2 -14870.472} C_VEL
LIN {X 0,Y 333.462,Z 727.368,A -85,B 0,C 180,E1 -14872.293,E2 -14872.293} C_VEL
LIN {X 0,Y 335.613,Z 716.517,A -85,B 0,C 180,E1 -14873.936,E2 -14873.936} C_VEL
LIN {X 0,Y 338.02,Z 703.571,A -85,B 0,C 180,E1 -14875.557,E2 -14875.557} C_VEL
LIN {X 0,Y 340.205,Z 690.759,A -85,B 0,C 180,E1 -14876.864,E2 -14876.864} C_VEL
LIN {X 0,Y 342.303,Z 676.428,A -85,B 0,C 180,E1 -14878.042,E2 -14878.042} C_VEL
LIN {X 0,Y 344.044,Z 662.446,A -85,B 0,C 180,E1 -14878.938,E2 -14878.938} C_VEL
LIN {X 0,Y 345.604,Z 647.794,A -85,B 0,C 180,E1 -14879.629,E2 -14879.629} C_VEL
LIN {X 0,Y 346.652,Z 633.039,A -85,B 0,C 180,E1 -14880.117,E2 -14880.117} C_VEL
LIN {X 0,Y 350.594,Z 519.127,A -85,B 0,C 180,E1 -14882.546,E2 -14882.546} C_VEL
LIN {X 0,Y 349,Z 507.905,A -85,B 0,C 180,E1 -14883.01,E2 -14883.01} C_VEL
LIN {X 0,Y 347.423,Z 500.142,A -85,B 0,C 180,E1 -14883.39,E2 -14883.39} C_VEL
LIN {X 0,Y 340.54,Z 484.853,A -85,B 0,C 180,E1 -14884.621,E2 -14884.621} C_VEL
LIN {X 0,Y 333.68,Z 471.421,A -85,B 0,C 180,E1 -14885.882,E2 -14885.882} C_VEL
LIN {X 0,Y 331.648,Z 467.348,A -85,B 0,C 180,E1 -14886.301,E2 -14886.301} C_VEL
LIN {X 0,Y 328.418,Z 456.246,A -85,B 0,C 180,E1 -14889.612,E2 -14889.612} C_VEL
LIN {X 0,Y 326.636,Z 450.427,A -85,B 0,C 180,E1 -14891.536,E2 -14891.536} C_VEL
LIN {X 0,Y 326.58,Z 450.43,A -85,B 0,C 180,E1 -14895.246,E2 -14895.246} C_VEL
LIN {X 0,Y 326.573,Z 450.433,A -85,B 0,C 180,E1 -14898.868,E2 -14898.868} C_VEL
LIN {X 0,Y 326.622,Z 450.425,A -85,B 0,C 180,E1 -14902.761,E2 -14902.761} C_VEL
LIN {X 0,Y 326.601,Z 450.429,A -85,B 0,C 180,E1 -14905.98,E2 -14905.98} C_VEL
LIN {X 0,Y 326.627,Z 450.421,A -85,B 0,C 180,E1 -14909.39,E2 -14909.39} C_VEL
LIN {X 0,Y 326.676,Z 450.411,A -85,B 0,C 180,E1 -14913.142,E2 -14913.142} C_VEL
LIN {X 0,Y 326.645,Z 450.417,A -85,B 0,C 180,E1 -14915.871,E2 -14915.871} C_VEL
LIN {X 0,Y 326.658,Z 450.413,A -85,B 0,C 180,E1 -14919.865,E2 -14919.865} C_VEL
LIN {X 0,Y 326.692,Z 450.41,A -85,B 0,C 180,E1 -14922.472,E2 -14922.472} C_VEL
LIN {X 0,Y 326.753,Z 450.402,A -85,B 0,C 180,E1 -14926.315,E2 -14926.315} C_VEL
LIN {X 0,Y 326.809,Z 450.395,A -85,B 0,C 180,E1 -14930.094,E2 -14930.094} C_VEL
LIN {X 0,Y 326.972,Z 450.381,A -85,B 0,C 180,E1 -14932.591,E2 -14932.591} C_VEL
LIN {X 0,Y 326.773,Z 450.404,A -85,B 0,C 180,E1 -14935.065,E2 -14935.065} C_VEL
LIN {X 0,Y 327.042,Z 450.365,A -85,B 0,C 180,E1 -14937.537,E2 -14937.537} C_VEL
LIN {X 0,Y 327.192,Z 450.355,A -85,B 0,C 180,E1 -14940,E2 -14940} C_VEL
LIN {X 0,Y 327.042,Z 450.37,A -85,B 0,C 180,E1 -14942.464,E2 -14942.464} C_VEL
LIN {X 0,Y 326.965,Z 450.378,A -85,B 0,C 180,E1 -14946.636,E2 -14946.636} C_VEL
LIN {X 0,Y 326.807,Z 450.403,A -85,B 0,C 180,E1 -14949.907,E2 -14949.907} C_VEL
LIN {X 0,Y 326.753,Z 450.405,A -85,B 0,C 180,E1 -14953.686,E2 -14953.686} C_VEL
LIN {X 0,Y 326.694,Z 450.415,A -85,B 0,C 180,E1 -14957.529,E2 -14957.529} C_VEL
LIN {X 0,Y 326.662,Z 450.421,A -85,B 0,C 180,E1 -14960.135,E2 -14960.135} C_VEL
LIN {X 0,Y 326.646,Z 450.425,A -85,B 0,C 180,E1 -14964.13,E2 -14964.13} C_VEL
LIN {X 0,Y 326.68,Z 450.41,A -85,B 0,C 180,E1 -14966.858,E2 -14966.858} C_VEL
LIN {X 0,Y 326.698,Z 450.576,A -85,B 0,C 180,E1 -14970.181,E2 -14970.181} C_VEL
LIN {X 0,Y 327.595,Z 453.616,A -85,B 0,C 180,E1 -14971.214,E2 -14971.214} C_VEL
LIN {X 0,Y 337.721,Z 471.267,A -85,B 0,C 180,E1 -14973.106,E2 -14973.106} C_VEL
LIN {X 0,Y 346.19,Z 487.971,A -85,B 0,C 180,E1 -14974.608,E2 -14974.608} C_VEL
LIN {X 0,Y 351.102,Z 498.981,A -85,B 0,C 180,E1 -14975.46,E2 -14975.46} C_VEL
LIN {X 0,Y 347.029,Z 617.677,A -85,B 0,C 180,E1 -14978.01,E2 -14978.01} C_VEL
LIN {X 0,Y 345.873,Z 633.368,A -85,B 0,C 180,E1 -14978.56,E2 -14978.56} C_VEL
LIN {X 0,Y 344.421,Z 648.646,A -85,B 0,C 180,E1 -14979.355,E2 -14979.355} C_VEL
LIN {X 0,Y 342.598,Z 663.581,A -85,B 0,C 180,E1 -14980.399,E2 -14980.399} C_VEL
LIN {X 0,Y 340.66,Z 676.972,A -85,B 0,C 180,E1 -14981.586,E2 -14981.586} C_VEL
LIN {X 0,Y 338.496,Z 689.589,A -85,B 0,C 180,E1 -14982.958,E2 -14982.958} C_VEL
LIN {X 0,Y 336.073,Z 702.501,A -85,B 0,C 180,E1 -14984.684,E2 -14984.684} C_VEL
LIN {X 0,Y 333.951,Z 713.259,A -85,B 0,C 180,E1 -14986.433,E2 -14986.433} C_VEL
LIN {X 0,Y 331.689,Z 723.991,A -85,B 0,C 180,E1 -14988.538,E2 -14988.538} C_VEL
LIN {X 0,Y 329.811,Z 732.876,A -85,B 0,C 180,E1 -14990.659,E2 -14990.659} C_VEL
LIN {X 0,Y 328.05,Z 741.355,A -85,B 0,C 180,E1 -14993.141,E2 -14993.141} C_VEL
LIN {X 0,Y 326.899,Z 747.391,A -85,B 0,C 180,E1 -14995.341,E2 -14995.341} C_VEL
LIN {X 0,Y 325.921,Z 753.371,A -85,B 0,C 180,E1 -14998.11,E2 -14998.11} C_VEL
LIN {X 0,Y 325.36,Z 756.764,A -85,B 0,C 180,E1 -15000.212,E2 -15000.212} C_VEL
LIN {X 0,Y 324.833,Z 759.938,A -85,B 0,C 180,E1 -15002.978,E2 -15002.978} C_VEL
LIN {X 0,Y 324.636,Z 761.651,A -85,B 0,C 180,E1 -15005.713,E2 -15005.713} C_VEL
LIN {X 0,Y 324.594,Z 761.965,A -85,B 0,C 180,E1 -15008.596,E2 -15008.596} C_VEL
LIN {X 0,Y 324.697,Z 761.027,A -85,B 0,C 180,E1 -15011.055,E2 -15011.055} C_VEL
LIN {X 0,Y 324.964,Z 758.79,A -85,B 0,C 180,E1 -15013.672,E2 -15013.672} C_VEL
LIN {X 0,Y 325.46,Z 755.119,A -85,B 0,C 180,E1 -15016.346,E2 -15016.346} C_VEL
LIN {X 0,Y 326.067,Z 750.432,A -85,B 0,C 180,E1 -15018.815,E2 -15018.815} C_VEL
LIN {X 0,Y 327.099,Z 744.147,A -85,B 0,C 180,E1 -15021.351,E2 -15021.351} C_VEL
LIN {X 0,Y 328.443,Z 736.267,A -85,B 0,C 180,E1 -15023.859,E2 -15023.859} C_VEL
LIN {X 0,Y 330.039,Z 727.861,A -85,B 0,C 180,E1 -15026.032,E2 -15026.032} C_VEL
LIN {X 0,Y 331.977,Z 717.743,A -85,B 0,C 180,E1 -15028.181,E2 -15028.181} C_VEL
LIN {X 0,Y 333.839,Z 707.455,A -85,B 0,C 180,E1 -15030.001,E2 -15030.001} C_VEL
LIN {X 0,Y 336.063,Z 695.103,A -85,B 0,C 180,E1 -15031.798,E2 -15031.798} C_VEL
LIN {X 0,Y 337.987,Z 683.621,A -85,B 0,C 180,E1 -15033.179,E2 -15033.179} C_VEL
LIN {X 0,Y 339.883,Z 670.861,A -85,B 0,C 180,E1 -15034.448,E2 -15034.448} C_VEL
LIN {X 0,Y 341.456,Z 658.364,A -85,B 0,C 180,E1 -15035.463,E2 -15035.463} C_VEL
LIN {X 0,Y 342.982,Z 643.805,A -85,B 0,C 180,E1 -15036.398,E2 -15036.398} C_VEL
LIN {X 0,Y 344.226,Z 628.758,A -85,B 0,C 180,E1 -15037.111,E2 -15037.111} C_VEL
LIN {X 0,Y 345.109,Z 613.105,A -85,B 0,C 180,E1 -15037.607,E2 -15037.607} C_VEL
LIN {X 0,Y 348.798,Z 497.601,A -85,B 0,C 180,E1 -15040.041,E2 -15040.041} C_VEL
LIN {X 0,Y 342.219,Z 482.285,A -85,B 0,C 180,E1 -15041.072,E2 -15041.072} C_VEL
LIN {X 0,Y 333.911,Z 465.26,A -85,B 0,C 180,E1 -15042.387,E2 -15042.387} C_VEL
LIN {X 0,Y 331.305,Z 460.099,A -85,B 0,C 180,E1 -15042.812,E2 -15042.812} C_VEL
LIN {X 0,Y 329.701,Z 458.783,A -85,B 0,C 180,E1 -15043.027,E2 -15043.027} C_VEL
LIN {X 0,Y 323.074,Z 456.937,A -85,B 0,C 180,E1 -15043.846,E2 -15043.846} C_VEL
LIN {X 0,Y 321.499,Z 455.615,A -85,B 0,C 180,E1 -15044.071,E2 -15044.071} C_VEL
LIN {X 0,Y 320.027,Z 452.578,A -85,B 0,C 180,E1 -15044.367,E2 -15044.367} C_VEL
LIN {X 0,Y 319.724,Z 451.285,A -85,B 0,C 180,E1 -15044.766,E2 -15044.766} C_VEL
LIN {X 0,Y 319.695,Z 451.288,A -85,B 0,C 180,E1 -15049.039,E2 -15049.039} C_VEL
LIN {X 0,Y 319.574,Z 451.301,A -85,B 0,C 180,E1 -15053.32,E2 -15053.32} C_VEL
LIN {X 0,Y 319.639,Z 451.296,A -85,B 0,C 180,E1 -15056.088,E2 -15056.088} C_VEL
LIN {X 0,Y 319.593,Z 451.293,A -85,B 0,C 180,E1 -15058.934,E2 -15058.934} C_VEL
LIN {X 0,Y 319.537,Z 451.297,A -85,B 0,C 180,E1 -15061.862,E2 -15061.862} C_VEL
LIN {X 0,Y 319.584,Z 451.304,A -85,B 0,C 180,E1 -15065.543,E2 -15065.543} C_VEL
LIN {X 0,Y 319.561,Z 451.288,A -85,B 0,C 180,E1 -15068.01,E2 -15068.01} C_VEL
LIN {X 0,Y 319.558,Z 451.304,A -85,B 0,C 180,E1 -15071.603,E2 -15071.603} C_VEL
LIN {X 0,Y 319.494,Z 451.311,A -85,B 0,C 180,E1 -15075.258,E2 -15075.258} C_VEL
LIN {X 0,Y 319.542,Z 451.293,A -85,B 0,C 180,E1 -15078.713,E2 -15078.713} C_VEL
LIN {X 0,Y 319.584,Z 451.296,A -85,B 0,C 180,E1 -15082.343,E2 -15082.343} C_VEL
LIN {X 0,Y 319.562,Z 451.294,A -85,B 0,C 180,E1 -15085.123,E2 -15085.123} C_VEL
LIN {X 0,Y 319.569,Z 451.295,A -85,B 0,C 180,E1 -15089.059,E2 -15089.059} C_VEL
LIN {X 0,Y 319.607,Z 451.296,A -85,B 0,C 180,E1 -15092.498,E2 -15092.498} C_VEL
LIN {X 0,Y 319.605,Z 451.29,A -85,B 0,C 180,E1 -15095.304,E2 -15095.304} C_VEL
LIN {X 0,Y 319.606,Z 451.296,A -85,B 0,C 180,E1 -15099.4,E2 -15099.4} C_VEL
LIN {X 0,Y 319.66,Z 451.28,A -85,B 0,C 180,E1 -15102.073,E2 -15102.073} C_VEL
LIN {X 0,Y 319.733,Z 451.283,A -85,B 0,C 180,E1 -15106.007,E2 -15106.007} C_VEL
LIN {X 0,Y 319.759,Z 451.261,A -85,B 0,C 180,E1 -15109.873,E2 -15109.873} C_VEL
LIN {X 0,Y 319.934,Z 451.254,A -85,B 0,C 180,E1 -15112.426,E2 -15112.426} C_VEL
LIN {X 0,Y 319.748,Z 451.277,A -85,B 0,C 180,E1 -15114.956,E2 -15114.956} C_VEL
LIN {X 0,Y 319.99,Z 451.233,A -85,B 0,C 180,E1 -15117.482,E2 -15117.482} C_VEL
LIN {X 0,Y 320.151,Z 451.232,A -85,B 0,C 180,E1 -15120,E2 -15120} C_VEL
LIN {X 0,Y 319.991,Z 451.241,A -85,B 0,C 180,E1 -15122.517,E2 -15122.517} C_VEL
LIN {X 0,Y 319.952,Z 451.245,A -85,B 0,C 180,E1 -15126.305,E2 -15126.305} C_VEL
LIN {X 0,Y 319.843,Z 451.267,A -85,B 0,C 180,E1 -15128.848,E2 -15128.848} C_VEL
LIN {X 0,Y 319.682,Z 451.271,A -85,B 0,C 180,E1 -15132.7,E2 -15132.7} C_VEL
LIN {X 0,Y 319.7,Z 451.286,A -85,B 0,C 180,E1 -15135.295,E2 -15135.295} C_VEL
LIN {X 0,Y 319.674,Z 451.273,A -85,B 0,C 180,E1 -15139.255,E2 -15139.255} C_VEL
LIN {X 0,Y 319.571,Z 451.3,A -85,B 0,C 180,E1 -15143.319,E2 -15143.319} C_VEL
LIN {X 0,Y 319.635,Z 451.294,A -85,B 0,C 180,E1 -15146.088,E2 -15146.088} C_VEL
LIN {X 0,Y 319.59,Z 451.297,A -85,B 0,C 180,E1 -15148.933,E2 -15148.933} C_VEL
LIN {X 0,Y 319.534,Z 451.308,A -85,B 0,C 180,E1 -15151.861,E2 -15151.861} C_VEL
LIN {X 0,Y 319.581,Z 451.3,A -85,B 0,C 180,E1 -15155.543,E2 -15155.543} C_VEL
LIN {X 0,Y 319.574,Z 451.3,A -85,B 0,C 180,E1 -15158.008,E2 -15158.008} C_VEL
LIN {X 0,Y 319.552,Z 451.307,A -85,B 0,C 180,E1 -15161.602,E2 -15161.602} C_VEL
LIN {X 0,Y 319.577,Z 451.304,A -85,B 0,C 180,E1 -15165.273,E2 -15165.273} C_VEL
LIN {X 0,Y 319.595,Z 451.301,A -85,B 0,C 180,E1 -15169.143,E2 -15169.143} C_VEL
LIN {X 0,Y 319.638,Z 451.48,A -85,B 0,C 180,E1 -15169.452,E2 -15169.452} C_VEL
LIN {X 0,Y 323.234,Z 464.312,A -85,B 0,C 180,E1 -15173.116,E2 -15173.116} C_VEL
LIN {X 0,Y 324.311,Z 468.436,A -85,B 0,C 180,E1 -15174.209,E2 -15174.209} C_VEL
LIN {X 0,Y 334.34,Z 489.831,A -85,B 0,C 180,E1 -15175.896,E2 -15175.896} C_VEL
LIN {X 0,Y 339.099,Z 500.893,A -85,B 0,C 180,E1 -15176.676,E2 -15176.676} C_VEL
LIN {X 0,Y 342.212,Z 518.951,A -85,B 0,C 180,E1 -15177.439,E2 -15177.439} C_VEL
LIN {X 0,Y 338.417,Z 634.588,A -85,B 0,C 180,E1 -15179.933,E2 -15179.933} C_VEL
LIN {X 0,Y 337.206,Z 650.786,A -85,B 0,C 180,E1 -15180.502,E2 -15180.502} C_VEL
LIN {X 0,Y 335.636,Z 666.036,A -85,B 0,C 180,E1 -15181.291,E2 -15181.291} C_VEL
LIN {X 0,Y 333.935,Z 679.832,A -85,B 0,C 180,E1 -15182.244,E2 -15182.244} C_VEL
LIN {X 0,Y 331.921,Z 693.392,A -85,B 0,C 180,E1 -15183.429,E2 -15183.429} C_VEL
LIN {X 0,Y 329.832,Z 705.867,A -85,B 0,C 180,E1 -15184.776,E2 -15184.776} C_VEL
LIN {X 0,Y 327.436,Z 718.553,A -85,B 0,C 180,E1 -15186.436,E2 -15186.436} C_VEL
LIN {X 0,Y 325.436,Z 729.37,A -85,B 0,C 180,E1 -15188.162,E2 -15188.162} C_VEL
LIN {X 0,Y 323.705,Z 739.044,A -85,B 0,C 180,E1 -15190.004,E2 -15190.004} C_VEL
LIN {X 0,Y 321.78,Z 748.69,A -85,B 0,C 180,E1 -15192.195,E2 -15192.195} C_VEL
LIN {X 0,Y 320.368,Z 756.726,A -85,B 0,C 180,E1 -15194.411,E2 -15194.411} C_VEL
LIN {X 0,Y 319.279,Z 763.397,A -85,B 0,C 180,E1 -15196.636,E2 -15196.636} C_VEL
LIN {X 0,Y 318.424,Z 769.514,A -85,B 0,C 180,E1 -15199.186,E2 -15199.186} C_VEL
LIN {X 0,Y 318.006,Z 774.207,A -85,B 0,C 180,E1 -15201.74,E2 -15201.74} C_VEL
LIN {X 0,Y 317.817,Z 777.626,A -85,B 0,C 180,E1 -15204.324,E2 -15204.324} C_VEL
LIN {X 0,Y 317.762,Z 779.335,A -85,B 0,C 180,E1 -15206.195,E2 -15206.195} C_VEL
LIN {X 0,Y 317.739,Z 780.607,A -85,B 0,C 180,E1 -15208.732,E2 -15208.732} C_VEL
LIN {X 0,Y 317.739,Z 780.686,A -85,B 0,C 180,E1 -15211.267,E2 -15211.267} C_VEL
LIN {X 0,Y 317.766,Z 779.616,A -85,B 0,C 180,E1 -15213.804,E2 -15213.804} C_VEL
LIN {X 0,Y 317.871,Z 777.387,A -85,B 0,C 180,E1 -15216.346,E2 -15216.346} C_VEL
LIN {X 0,Y 318.097,Z 773.954,A -85,B 0,C 180,E1 -15218.896,E2 -15218.896} C_VEL
LIN {X 0,Y 318.631,Z 769.23,A -85,B 0,C 180,E1 -15221.449,E2 -15221.449} C_VEL
LIN {X 0,Y 319.595,Z 763.088,A -85,B 0,C 180,E1 -15223.997,E2 -15223.997} C_VEL
LIN {X 0,Y 321.026,Z 755.403,A -85,B 0,C 180,E1 -15226.534,E2 -15226.534} C_VEL
LIN {X 0,Y 322.646,Z 747.197,A -85,B 0,C 180,E1 -15228.74,E2 -15228.74} C_VEL
LIN {X 0,Y 324.864,Z 737.379,A -85,B 0,C 180,E1 -15230.912,E2 -15230.912} C_VEL
LIN {X 0,Y 326.857,Z 727.354,A -85,B 0,C 180,E1 -15232.769,E2 -15232.769} C_VEL
LIN {X 0,Y 329.119,Z 716.542,A -85,B 0,C 180,E1 -15234.439,E2 -15234.439} C_VEL
LIN {X 0,Y 331.617,Z 703.644,A -85,B 0,C 180,E1 -15236.087,E2 -15236.087} C_VEL
LIN {X 0,Y 333.898,Z 690.895,A -85,B 0,C 180,E1 -15237.414,E2 -15237.414} C_VEL
LIN {X 0,Y 336.016,Z 676.975,A -85,B 0,C 180,E1 -15238.587,E2 -15238.587} C_VEL
LIN {X 0,Y 337.863,Z 662.822,A -85,B 0,C 180,E1 -15239.519,E2 -15239.519} C_VEL
LIN {X 0,Y 339.495,Z 648.439,A -85,B 0,C 180,E1 -15240.217,E2 -15240.217} C_VEL
LIN {X 0,Y 340.584,Z 634.244,A -85,B 0,C 180,E1 -15240.711,E2 -15240.711} C_VEL
LIN {X 0,Y 344.741,Z 519.649,A -85,B 0,C 180,E1 -15243.201,E2 -15243.201} C_VEL
LIN {X 0,Y 342.206,Z 504.142,A -85,B 0,C 180,E1 -15243.905,E2 -15243.905} C_VEL
LIN {X 0,Y 338.709,Z 495.565,A -85,B 0,C 180,E1 -15244.565,E2 -15244.565} C_VEL
LIN {X 0,Y 330.369,Z 478.476,A -85,B 0,C 180,E1 -15246.135,E2 -15246.135} C_VEL
LIN {X 0,Y 324.337,Z 467.072,A -85,B 0,C 180,E1 -15247.352,E2 -15247.352} C_VEL
LIN {X 0,Y 321.055,Z 455.985,A -85,B 0,C 180,E1 -15250.832,E2 -15250.832} C_VEL
LIN {X 0,Y 319.565,Z 451.296,A -85,B 0,C 180,E1 -15252.427,E2 -15252.427} C_VEL
LIN {X 0,Y 319.538,Z 451.307,A -85,B 0,C 180,E1 -15255.266,E2 -15255.266} C_VEL
LIN {X 0,Y 319.524,Z 451.312,A -85,B 0,C 180,E1 -15258.711,E2 -15258.711} C_VEL
LIN {X 0,Y 319.556,Z 451.303,A -85,B 0,C 180,E1 -15262.347,E2 -15262.347} C_VEL
LIN {X 0,Y 319.554,Z 451.304,A -85,B 0,C 180,E1 -15265.123,E2 -15265.123} C_VEL
LIN {X 0,Y 319.56,Z 451.303,A -85,B 0,C 180,E1 -15269.059,E2 -15269.059} C_VEL
LIN {X 0,Y 319.598,Z 451.294,A -85,B 0,C 180,E1 -15272.497,E2 -15272.497} C_VEL
LIN {X 0,Y 319.598,Z 451.298,A -85,B 0,C 180,E1 -15275.304,E2 -15275.304} C_VEL
LIN {X 0,Y 319.59,Z 451.302,A -85,B 0,C 180,E1 -15278.048,E2 -15278.048} C_VEL
LIN {X 0,Y 319.682,Z 451.289,A -85,B 0,C 180,E1 -15280.962,E2 -15280.962} C_VEL
LIN {X 0,Y 319.724,Z 451.283,A -85,B 0,C 180,E1 -15285.276,E2 -15285.276} C_VEL
LIN {X 0,Y 319.753,Z 451.275,A -85,B 0,C 180,E1 -15289.873,E2 -15289.873} C_VEL
LIN {X 0,Y 319.926,Z 451.26,A -85,B 0,C 180,E1 -15292.426,E2 -15292.426} C_VEL
LIN {X 0,Y 319.743,Z 451.278,A -85,B 0,C 180,E1 -15294.956,E2 -15294.956} C_VEL
LIN {X 0,Y 319.986,Z 451.244,A -85,B 0,C 180,E1 -15297.483,E2 -15297.483} C_VEL
LIN {X 0,Y 320.144,Z 451.233,A -85,B 0,C 180,E1 -15300,E2 -15300} C_VEL
LIN {X 0,Y 319.986,Z 451.25,A -85,B 0,C 180,E1 -15302.518,E2 -15302.518} C_VEL
LIN {X 0,Y 319.926,Z 451.257,A -85,B 0,C 180,E1 -15306.626,E2 -15306.626} C_VEL
LIN {X 0,Y 319.751,Z 451.28,A -85,B 0,C 180,E1 -15310.128,E2 -15310.128} C_VEL
LIN {X 0,Y 319.725,Z 451.282,A -85,B 0,C 180,E1 -15314.725,E2 -15314.725} C_VEL
LIN {X 0,Y 319.684,Z 451.286,A -85,B 0,C 180,E1 -15319.039,E2 -15319.039} C_VEL
LIN {X 0,Y 319.565,Z 451.306,A -85,B 0,C 180,E1 -15323.32,E2 -15323.32} C_VEL
LIN {X 0,Y 319.63,Z 451.288,A -85,B 0,C 180,E1 -15326.089,E2 -15326.089} C_VEL
LIN {X 0,Y 319.613,Z 451.297,A -85,B 0,C 180,E1 -15329.202,E2 -15329.202} C_VEL
LIN {X 0,Y 320.47,Z 454.089,A -85,B 0,C 180,E1 -15330.155,E2 -15330.155} C_VEL
LIN {X 0,Y 322.53,Z 457.622,A -85,B 0,C 180,E1 -15330.579,E2 -15330.579} C_VEL
LIN {X 0,Y 331.1,Z 472.192,A -85,B 0,C 180,E1 -15332.245,E2 -15332.245} C_VEL
LIN {X 0,Y 339.6,Z 488.713,A -85,B 0,C 180,E1 -15333.82,E2 -15333.82} C_VEL
LIN {X 0,Y 345.222,Z 501.184,A -85,B 0,C 180,E1 -15334.835,E2 -15334.835} C_VEL
LIN {X 0,Y 341.036,Z 617.7,A -85,B 0,C 180,E1 -15337.376,E2 -15337.376} C_VEL
LIN {X 0,Y 339.793,Z 633.871,A -85,B 0,C 180,E1 -15337.952,E2 -15337.952} C_VEL
LIN {X 0,Y 338.301,Z 648.994,A -85,B 0,C 180,E1 -15338.756,E2 -15338.756} C_VEL
LIN {X 0,Y 336.443,Z 663.642,A -85,B 0,C 180,E1 -15339.795,E2 -15339.795} C_VEL
LIN {X 0,Y 334.333,Z 677.567,A -85,B 0,C 180,E1 -15341.053,E2 -15341.053} C_VEL
LIN {X 0,Y 332.158,Z 689.774,A -85,B 0,C 180,E1 -15342.403,E2 -15342.403} C_VEL
LIN {X 0,Y 329.601,Z 702.766,A -85,B 0,C 180,E1 -15344.169,E2 -15344.169} C_VEL
LIN {X 0,Y 327.579,Z 712.627,A -85,B 0,C 180,E1 -15345.794,E2 -15345.794} C_VEL
LIN {X 0,Y 325.171,Z 723.509,A -85,B 0,C 180,E1 -15347.934,E2 -15347.934} C_VEL
LIN {X 0,Y 323.173,Z 732.499,A -85,B 0,C 180,E1 -15350.095,E2 -15350.095} C_VEL
LIN {X 0,Y 321.545,Z 739.954,A -85,B 0,C 180,E1 -15352.267,E2 -15352.267} C_VEL
LIN {X 0,Y 320.131,Z 746.809,A -85,B 0,C 180,E1 -15354.715,E2 -15354.715} C_VEL
LIN {X 0,Y 319.022,Z 752.749,A -85,B 0,C 180,E1 -15357.424,E2 -15357.424} C_VEL
LIN {X 0,Y 318.47,Z 756.274,A -85,B 0,C 180,E1 -15359.5,E2 -15359.5} C_VEL
LIN {X 0,Y 317.86,Z 759.715,A -85,B 0,C 180,E1 -15362.335,E2 -15362.335} C_VEL
LIN {X 0,Y 317.555,Z 761.686,A -85,B 0,C 180,E1 -15365.149,E2 -15365.149} C_VEL
LIN {X 0,Y 317.453,Z 762.267,A -85,B 0,C 180,E1 -15367.893,E2 -15367.893} C_VEL
LIN {X 0,Y 317.567,Z 761.532,A -85,B 0,C 180,E1 -15370.613,E2 -15370.613} C_VEL
LIN {X 0,Y 317.826,Z 759.505,A -85,B 0,C 180,E1 -15373.295,E2 -15373.295} C_VEL
LIN {X 0,Y 318.273,Z 756.193,A -85,B 0,C 180,E1 -15375.943,E2 -15375.943} C_VEL
LIN {X 0,Y 318.892,Z 751.579,A -85,B 0,C 180,E1 -15378.56,E2 -15378.56} C_VEL
LIN {X 0,Y 319.972,Z 745.268,A -85,B 0,C 180,E1 -15381.266,E2 -15381.266} C_VEL
LIN {X 0,Y 321.276,Z 737.981,A -85,B 0,C 180,E1 -15383.721,E2 -15383.721} C_VEL
LIN {X 0,Y 322.84,Z 729.861,A -85,B 0,C 180,E1 -15385.944,E2 -15385.944} C_VEL
LIN {X 0,Y 324.786,Z 720.117,A -85,B 0,C 180,E1 -15388.141,E2 -15388.141} C_VEL
LIN {X 0,Y 326.719,Z 710.173,A -85,B 0,C 180,E1 -15390.001,E2 -15390.001} C_VEL
LIN {X 0,Y 328.921,Z 698.361,A -85,B 0,C 180,E1 -15391.837,E2 -15391.837} C_VEL
LIN {X 0,Y 331.074,Z 686.194,A -85,B 0,C 180,E1 -15393.394,E2 -15393.394} C_VEL
LIN {X 0,Y 333.241,Z 672.348,A -85,B 0,C 180,E1 -15394.84,E2 -15394.84} C_VEL
LIN {X 0,Y 335.129,Z 658.173,A -85,B 0,C 180,E1 -15396.019,E2 -15396.019} C_VEL
LIN {X 0,Y 336.707,Z 643.488,A -85,B 0,C 180,E1 -15396.969,E2 -15396.969} C_VEL
LIN {X 0,Y 337.99,Z 628.23,A -85,B 0,C 180,E1 -15397.693,E2 -15397.693} C_VEL
LIN {X 0,Y 338.849,Z 613.558,A -85,B 0,C 180,E1 -15398.161,E2 -15398.161} C_VEL
LIN {X 0,Y 342.567,Z 499.302,A -85,B 0,C 180,E1 -15400.615,E2 -15400.615} C_VEL
LIN {X 0,Y 335.135,Z 482.225,A -85,B 0,C 180,E1 -15401.817,E2 -15401.817} C_VEL
LIN {X 0,Y 325.905,Z 463.762,A -85,B 0,C 180,E1 -15403.33,E2 -15403.33} C_VEL
LIN {X 0,Y 321.499,Z 455.615,A -85,B 0,C 180,E1 -15404.071,E2 -15404.071} C_VEL
LIN {X 0,Y 319.586,Z 453.505,A -85,B 0,C 180,E1 -15404.485,E2 -15404.485} C_VEL
LIN {X 0,Y 317.812,Z 452.374,A -85,B 0,C 180,E1 -15405.041,E2 -15405.041} C_VEL
LIN {X 0,Y 315.604,Z 451.86,A -85,B 0,C 180,E1 -15406.018,E2 -15406.018} C_VEL
LIN {X 0,Y 313.271,Z 452.084,A -85,B 0,C 180,E1 -15407.889,E2 -15407.889} C_VEL
LIN {X 0,Y 312.622,Z 452.171,A -85,B 0,C 180,E1 -15409.455,E2 -15409.455} C_VEL
LIN {X 0,Y 312.55,Z 452.18,A -85,B 0,C 180,E1 -15412.79,E2 -15412.79} C_VEL
LIN {X 0,Y 312.607,Z 452.173,A -85,B 0,C 180,E1 -15415.936,E2 -15415.936} C_VEL
LIN {X 0,Y 312.549,Z 452.176,A -85,B 0,C 180,E1 -15419.65,E2 -15419.65} C_VEL
LIN {X 0,Y 312.523,Z 452.172,A -85,B 0,C 180,E1 -15423.689,E2 -15423.689} C_VEL
LIN {X 0,Y 312.529,Z 452.166,A -85,B 0,C 180,E1 -15427.385,E2 -15427.385} C_VEL
LIN {X 0,Y 312.495,Z 452.183,A -85,B 0,C 180,E1 -15430.709,E2 -15430.709} C_VEL
LIN {X 0,Y 312.455,Z 452.184,A -85,B 0,C 180,E1 -15434.209,E2 -15434.209} C_VEL
LIN {X 0,Y 312.524,Z 452.168,A -85,B 0,C 180,E1 -15437.911,E2 -15437.911} C_VEL
LIN {X 0,Y 312.546,Z 452.176,A -85,B 0,C 180,E1 -15441.908,E2 -15441.908} C_VEL
LIN {X 0,Y 312.509,Z 452.178,A -85,B 0,C 180,E1 -15445.79,E2 -15445.79} C_VEL
LIN {X 0,Y 312.523,Z 452.175,A -85,B 0,C 180,E1 -15448.853,E2 -15448.853} C_VEL
LIN {X 0,Y 312.572,Z 452.168,A -85,B 0,C 180,E1 -15451.824,E2 -15451.824} C_VEL
LIN {X 0,Y 312.587,Z 452.168,A -85,B 0,C 180,E1 -15454.711,E2 -15454.711} C_VEL
LIN {X 0,Y 312.541,Z 452.174,A -85,B 0,C 180,E1 -15458.913,E2 -15458.913} C_VEL
LIN {X 0,Y 312.64,Z 452.158,A -85,B 0,C 180,E1 -15461.656,E2 -15461.656} C_VEL
LIN {X 0,Y 312.695,Z 452.155,A -85,B 0,C 180,E1 -15465.686,E2 -15465.686} C_VEL
LIN {X 0,Y 312.703,Z 452.141,A -85,B 0,C 180,E1 -15469.642,E2 -15469.642} C_VEL
LIN {X 0,Y 312.873,Z 452.134,A -85,B 0,C 180,E1 -15472.254,E2 -15472.254} C_VEL
LIN {X 0,Y 312.719,Z 452.153,A -85,B 0,C 180,E1 -15474.842,E2 -15474.842} C_VEL
LIN {X 0,Y 312.991,Z 452.115,A -85,B 0,C 180,E1 -15478.713,E2 -15478.713} C_VEL
LIN {X 0,Y 312.991,Z 452.123,A -85,B 0,C 180,E1 -15481.286,E2 -15481.286} C_VEL
LIN {X 0,Y 312.717,Z 452.131,A -85,B 0,C 180,E1 -15485.157,E2 -15485.157} C_VEL
LIN {X 0,Y 312.873,Z 452.137,A -85,B 0,C 180,E1 -15487.745,E2 -15487.745} C_VEL
LIN {X 0,Y 312.669,Z 452.142,A -85,B 0,C 180,E1 -15491.671,E2 -15491.671} C_VEL
LIN {X 0,Y 312.7,Z 452.156,A -85,B 0,C 180,E1 -15494.887,E2 -15494.887} C_VEL
LIN {X 0,Y 312.63,Z 452.15,A -85,B 0,C 180,E1 -15499.236,E2 -15499.236} C_VEL
LIN {X 0,Y 312.546,Z 452.174,A -85,B 0,C 180,E1 -15502.789,E2 -15502.789} C_VEL
LIN {X 0,Y 312.603,Z 452.169,A -85,B 0,C 180,E1 -15505.935,E2 -15505.935} C_VEL
LIN {X 0,Y 312.545,Z 452.179,A -85,B 0,C 180,E1 -15509.65,E2 -15509.65} C_VEL
LIN {X 0,Y 312.52,Z 452.179,A -85,B 0,C 180,E1 -15513.689,E2 -15513.689} C_VEL
LIN {X 0,Y 312.538,Z 452.18,A -85,B 0,C 180,E1 -15517.383,E2 -15517.383} C_VEL
LIN {X 0,Y 312.49,Z 452.184,A -85,B 0,C 180,E1 -15520.709,E2 -15520.709} C_VEL
LIN {X 0,Y 312.51,Z 452.181,A -85,B 0,C 180,E1 -15524.199,E2 -15524.199} C_VEL
LIN {X 0,Y 312.552,Z 452.176,A -85,B 0,C 180,E1 -15528.212,E2 -15528.212} C_VEL
LIN {X 0,Y 312.582,Z 452.347,A -85,B 0,C 180,E1 -15528.723,E2 -15528.723} C_VEL
LIN {X 0,Y 315.898,Z 463.978,A -85,B 0,C 180,E1 -15532.165,E2 -15532.165} C_VEL
LIN {X 0,Y 317.025,Z 468.16,A -85,B 0,C 180,E1 -15533.329,E2 -15533.329} C_VEL
LIN {X 0,Y 327.071,Z 489.257,A -85,B 0,C 180,E1 -15535.082,E2 -15535.082} C_VEL
LIN {X 0,Y 333.276,Z 503.493,A -85,B 0,C 180,E1 -15536.133,E2 -15536.133} C_VEL
LIN {X 0,Y 336.066,Z 520.317,A -85,B 0,C 180,E1 -15536.854,E2 -15536.854} C_VEL
LIN {X 0,Y 332.101,Z 635.516,A -85,B 0,C 180,E1 -15539.388,E2 -15539.388} C_VEL
LIN {X 0,Y 330.847,Z 651.274,A -85,B 0,C 180,E1 -15539.965,E2 -15539.965} C_VEL
LIN {X 0,Y 329.235,Z 666.522,A -85,B 0,C 180,E1 -15540.78,E2 -15540.78} C_VEL
LIN {X 0,Y 327.324,Z 681.001,A -85,B 0,C 180,E1 -15541.812,E2 -15541.812} C_VEL
LIN {X 0,Y 325.28,Z 694.323,A -85,B 0,C 180,E1 -15543.017,E2 -15543.017} C_VEL
LIN {X 0,Y 322.919,Z 707.872,A -85,B 0,C 180,E1 -15544.542,E2 -15544.542} C_VEL
LIN {X 0,Y 320.453,Z 720.192,A -85,B 0,C 180,E1 -15546.234,E2 -15546.234} C_VEL
LIN {X 0,Y 318.193,Z 731.908,A -85,B 0,C 180,E1 -15548.211,E2 -15548.211} C_VEL
LIN {X 0,Y 316.345,Z 741.664,A -85,B 0,C 180,E1 -15550.196,E2 -15550.196} C_VEL
LIN {X 0,Y 314.472,Z 750.837,A -85,B 0,C 180,E1 -15552.439,E2 -15552.439} C_VEL
LIN {X 0,Y 312.914,Z 759.262,A -85,B 0,C 180,E1 -15554.966,E2 -15554.966} C_VEL
LIN {X 0,Y 311.841,Z 766.355,A -85,B 0,C 180,E1 -15557.637,E2 -15557.637} C_VEL
LIN {X 0,Y 311.143,Z 771.76,A -85,B 0,C 180,E1 -15560.246,E2 -15560.246} C_VEL
LIN {X 0,Y 310.841,Z 774.891,A -85,B 0,C 180,E1 -15562.203,E2 -15562.203} C_VEL
LIN {X 0,Y 310.683,Z 778.005,A -85,B 0,C 180,E1 -15564.808,E2 -15564.808} C_VEL
LIN {X 0,Y 310.666,Z 779.904,A -85,B 0,C 180,E1 -15567.406,E2 -15567.406} C_VEL
LIN {X 0,Y 310.69,Z 780.58,A -85,B 0,C 180,E1 -15569.999,E2 -15569.999} C_VEL
LIN {X 0,Y 310.668,Z 780.099,A -85,B 0,C 180,E1 -15572.592,E2 -15572.592} C_VEL
LIN {X 0,Y 310.684,Z 778.466,A -85,B 0,C 180,E1 -15575.191,E2 -15575.191} C_VEL
LIN {X 0,Y 310.841,Z 775.656,A -85,B 0,C 180,E1 -15577.796,E2 -15577.796} C_VEL
LIN {X 0,Y 311.283,Z 771.61,A -85,B 0,C 180,E1 -15580.405,E2 -15580.405} C_VEL
LIN {X 0,Y 312.136,Z 766.207,A -85,B 0,C 180,E1 -15583.011,E2 -15583.011} C_VEL
LIN {X 0,Y 313.318,Z 759.339,A -85,B 0,C 180,E1 -15585.614,E2 -15585.614} C_VEL
LIN {X 0,Y 315.096,Z 750.831,A -85,B 0,C 180,E1 -15588.195,E2 -15588.195} C_VEL
LIN {X 0,Y 317.177,Z 741.769,A -85,B 0,C 180,E1 -15590.424,E2 -15590.424} C_VEL
LIN {X 0,Y 319.2,Z 732.29,A -85,B 0,C 180,E1 -15592.372,E2 -15592.372} C_VEL
LIN {X 0,Y 321.487,Z 721.683,A -85,B 0,C 180,E1 -15594.197,E2 -15594.197} C_VEL
LIN {X 0,Y 323.98,Z 709.869,A -85,B 0,C 180,E1 -15595.884,E2 -15595.884} C_VEL
LIN {X 0,Y 326.532,Z 696.995,A -85,B 0,C 180,E1 -15597.39,E2 -15597.39} C_VEL
LIN {X 0,Y 328.992,Z 682.691,A -85,B 0,C 180,E1 -15598.74,E2 -15598.74} C_VEL
LIN {X 0,Y 331.108,Z 667.968,A -85,B 0,C 180,E1 -15599.832,E2 -15599.832} C_VEL
LIN {X 0,Y 332.916,Z 653.05,A -85,B 0,C 180,E1 -15600.659,E2 -15600.659} C_VEL
LIN {X 0,Y 334.365,Z 637.547,A -85,B 0,C 180,E1 -15601.258,E2 -15601.258} C_VEL
LIN {X 0,Y 335.281,Z 616.656,A -85,B 0,C 180,E1 -15601.779,E2 -15601.779} C_VEL
LIN {X 0,Y 338.261,Z 536.709,A -85,B 0,C 180,E1 -15603.523,E2 -15603.523} C_VEL
LIN {X 0,Y 338.836,Z 519.851,A -85,B 0,C 180,E1 -15603.9,E2 -15603.9} C_VEL
LIN {X 0,Y 336.537,Z 506.157,A -85,B 0,C 180,E1 -15604.554,E2 -15604.554} C_VEL
LIN {X 0,Y 330.423,Z 492.47,A -85,B 0,C 180,E1 -15605.734,E2 -15605.734} C_VEL
LIN {X 0,Y 323.943,Z 479.563,A -85,B 0,C 180,E1 -15607.018,E2 -15607.018} C_VEL
LIN {X 0,Y 318.873,Z 470.435,A -85,B 0,C 180,E1 -15608.053,E2 -15608.053} C_VEL
LIN {X 0,Y 316.999,Z 466.739,A -85,B 0,C 180,E1 -15608.495,E2 -15608.495} C_VEL
LIN {X 0,Y 314.242,Z 457.673,A -85,B 0,C 180,E1 -15611.478,E2 -15611.478} C_VEL
LIN {X 0,Y 312.555,Z 452.169,A -85,B 0,C 180,E1 -15613.46,E2 -15613.46} C_VEL
LIN {X 0,Y 312.512,Z 452.175,A -85,B 0,C 180,E1 -15617.572,E2 -15617.572} C_VEL
LIN {X 0,Y 312.497,Z 452.186,A -85,B 0,C 180,E1 -15620.971,E2 -15620.971} C_VEL
LIN {X 0,Y 312.526,Z 452.177,A -85,B 0,C 180,E1 -15624.22,E2 -15624.22} C_VEL
LIN {X 0,Y 312.498,Z 452.179,A -85,B 0,C 180,E1 -15627.333,E2 -15627.333} C_VEL
LIN {X 0,Y 312.538,Z 452.179,A -85,B 0,C 180,E1 -15631.278,E2 -15631.278} C_VEL
LIN {X 0,Y 312.578,Z 452.174,A -85,B 0,C 180,E1 -15634.711,E2 -15634.711} C_VEL
LIN {X 0,Y 312.58,Z 452.173,A -85,B 0,C 180,E1 -15637.529,E2 -15637.529} C_VEL
LIN {X 0,Y 312.631,Z 452.168,A -85,B 0,C 180,E1 -15641.656,E2 -15641.656} C_VEL
LIN {X 0,Y 312.687,Z 452.159,A -85,B 0,C 180,E1 -15645.686,E2 -15645.686} C_VEL
LIN {X 0,Y 312.697,Z 452.155,A -85,B 0,C 180,E1 -15649.642,E2 -15649.642} C_VEL
LIN {X 0,Y 312.865,Z 452.14,A -85,B 0,C 180,E1 -15652.254,E2 -15652.254} C_VEL
LIN {X 0,Y 312.713,Z 452.152,A -85,B 0,C 180,E1 -15654.843,E2 -15654.843} C_VEL
LIN {X 0,Y 312.984,Z 452.12,A -85,B 0,C 180,E1 -15658.714,E2 -15658.714} C_VEL
LIN {X 0,Y 312.984,Z 452.114,A -85,B 0,C 180,E1 -15661.287,E2 -15661.287} C_VEL
LIN {X 0,Y 312.713,Z 452.151,A -85,B 0,C 180,E1 -15665.158,E2 -15665.158} C_VEL
LIN {X 0,Y 312.865,Z 452.133,A -85,B 0,C 180,E1 -15667.746,E2 -15667.746} C_VEL
LIN {X 0,Y 312.663,Z 452.159,A -85,B 0,C 180,E1 -15671.672,E2 -15671.672} C_VEL
LIN {X 0,Y 312.694,Z 452.159,A -85,B 0,C 180,E1 -15674.888,E2 -15674.888} C_VEL
LIN {X 0,Y 312.626,Z 452.165,A -85,B 0,C 180,E1 -15679.238,E2 -15679.238} C_VEL
LIN {X 0,Y 312.54,Z 452.183,A -85,B 0,C 180,E1 -15682.79,E2 -15682.79} C_VEL
LIN {X 0,Y 312.598,Z 452.165,A -85,B 0,C 180,E1 -15685.936,E2 -15685.936} C_VEL
LIN {X 0,Y 312.601,Z 452.356,A -85,B 0,C 180,E1 -15688.281,E2 -15688.281} C_VEL
LIN {X 0,Y 313.208,Z 454.332,A -85,B 0,C 180,E1 -15688.991,E2 -15688.991} C_VEL
LIN {X 0,Y 315.785,Z 458.489,A -85,B 0,C 180,E1 -15689.545,E2 -15689.545} C_VEL
LIN {X 0,Y 323.766,Z 471.864,A -85,B 0,C 180,E1 -15691.187,E2 -15691.187} C_VEL
LIN {X 0,Y 331.404,Z 486.076,A -85,B 0,C 180,E1 -15692.676,E2 -15692.676} C_VEL
LIN {X 0,Y 338.917,Z 502.095,A -85,B 0,C 180,E1 -15694.093,E2 -15694.093} C_VEL
LIN {X 0,Y 339.401,Z 503.615,A -85,B 0,C 180,E1 -15694.195,E2 -15694.195} C_VEL
LIN {X 0,Y 335.095,Z 617.842,A -85,B 0,C 180,E1 -15696.722,E2 -15696.722} C_VEL
LIN {X 0,Y 333.832,Z 633.541,A -85,B 0,C 180,E1 -15697.28,E2 -15697.28} C_VEL
LIN {X 0,Y 332.353,Z 648.221,A -85,B 0,C 180,E1 -15698.059,E2 -15698.059} C_VEL
LIN {X 0,Y 330.492,Z 662.79,A -85,B 0,C 180,E1 -15699.09,E2 -15699.09} C_VEL
LIN {X 0,Y 328.313,Z 676.393,A -85,B 0,C 180,E1 -15700.308,E2 -15700.308} C_VEL
LIN {X 0,Y 326.084,Z 688.633,A -85,B 0,C 180,E1 -15701.664,E2 -15701.664} C_VEL
LIN {X 0,Y 323.619,Z 700.945,A -85,B 0,C 180,E1 -15703.323,E2 -15703.323} C_VEL
LIN {X 0,Y 321.229,Z 711.984,A -85,B 0,C 180,E1 -15705.125,E2 -15705.125} C_VEL
LIN {X 0,Y 319.106,Z 721.317,A -85,B 0,C 180,E1 -15706.943,E2 -15706.943} C_VEL
LIN {X 0,Y 317.1,Z 729.809,A -85,B 0,C 180,E1 -15708.9,E2 -15708.9} C_VEL
LIN {X 0,Y 315.106,Z 738.55,A -85,B 0,C 180,E1 -15711.356,E2 -15711.356} C_VEL
LIN {X 0,Y 313.555,Z 745.588,A -85,B 0,C 180,E1 -15713.795,E2 -15713.795} C_VEL
LIN {X 0,Y 312.301,Z 751.505,A -85,B 0,C 180,E1 -15716.372,E2 -15716.372} C_VEL
LIN {X 0,Y 311.524,Z 756.114,A -85,B 0,C 180,E1 -15719.013,E2 -15719.013} C_VEL
LIN {X 0,Y 310.837,Z 759.641,A -85,B 0,C 180,E1 -15721.86,E2 -15721.86} C_VEL
LIN {X 0,Y 310.48,Z 761.835,A -85,B 0,C 180,E1 -15724.883,E2 -15724.883} C_VEL
LIN {X 0,Y 310.367,Z 762.452,A -85,B 0,C 180,E1 -15727.36,E2 -15727.36} C_VEL
LIN {X 0,Y 310.445,Z 761.932,A -85,B 0,C 180,E1 -15730.15,E2 -15730.15} C_VEL
LIN {X 0,Y 310.695,Z 760.13,A -85,B 0,C 180,E1 -15732.9,E2 -15732.9} C_VEL
LIN {X 0,Y 311.099,Z 757.058,A -85,B 0,C 180,E1 -15735.612,E2 -15735.612} C_VEL
LIN {X 0,Y 311.734,Z 752.684,A -85,B 0,C 180,E1 -15738.294,E2 -15738.294} C_VEL
LIN {X 0,Y 312.726,Z 746.92,A -85,B 0,C 180,E1 -15740.95,E2 -15740.95} C_VEL
LIN {X 0,Y 314.085,Z 739.628,A -85,B 0,C 180,E1 -15743.577,E2 -15743.577} C_VEL
LIN {X 0,Y 315.595,Z 731.834,A -85,B 0,C 180,E1 -15745.85,E2 -15745.85} C_VEL
LIN {X 0,Y 317.613,Z 722.419,A -85,B 0,C 180,E1 -15748.099,E2 -15748.099} C_VEL
LIN {X 0,Y 319.598,Z 712.866,A -85,B 0,C 180,E1 -15750.001,E2 -15750.001} C_VEL
LIN {X 0,Y 321.776,Z 701.553,A -85,B 0,C 180,E1 -15751.878,E2 -15751.878} C_VEL
LIN {X 0,Y 324.098,Z 689.04,A -85,B 0,C 180,E1 -15753.582,E2 -15753.582} C_VEL
LIN {X 0,Y 326.4,Z 675.333,A -85,B 0,C 180,E1 -15755.096,E2 -15755.096} C_VEL
LIN {X 0,Y 328.341,Z 661.849,A -85,B 0,C 180,E1 -15756.299,E2 -15756.299} C_VEL
LIN {X 0,Y 330.089,Z 646.924,A -85,B 0,C 180,E1 -15757.34,E2 -15757.34} C_VEL
LIN {X 0,Y 331.482,Z 632.047,A -85,B 0,C 180,E1 -15758.113,E2 -15758.113} C_VEL
LIN {X 0,Y 332.53,Z 616.647,A -85,B 0,C 180,E1 -15758.661,E2 -15758.661} C_VEL
LIN {X 0,Y 336.475,Z 501.249,A -85,B 0,C 180,E1 -15761.19,E2 -15761.19} C_VEL
LIN {X 0,Y 328.339,Z 482.887,A -85,B 0,C 180,E1 -15762.546,E2 -15762.546} C_VEL
LIN {X 0,Y 318.553,Z 463.632,A -85,B 0,C 180,E1 -15764.21,E2 -15764.21} C_VEL
LIN {X 0,Y 314.029,Z 455.475,A -85,B 0,C 180,E1 -15765.004,E2 -15765.004} C_VEL
LIN {X 0,Y 312.802,Z 452.818,A -85,B 0,C 180,E1 -15765.264,E2 -15765.264} C_VEL
LIN {X 0,Y 312.662,Z 452.16,A -85,B 0,C 180,E1 -15765.515,E2 -15765.515} C_VEL
LIN {X 0,Y 312.622,Z 452.171,A -85,B 0,C 180,E1 -15769.455,E2 -15769.455} C_VEL
LIN {X 0,Y 311.908,Z 452.263,A -85,B 0,C 180,E1 -15770.53,E2 -15770.53} C_VEL
LIN {X 0,Y 309.008,Z 452.622,A -85,B 0,C 180,E1 -15772.279,E2 -15772.279} C_VEL
LIN {X 0,Y 306.592,Z 452.914,A -85,B 0,C 180,E1 -15773.698,E2 -15773.698} C_VEL
LIN {X 0,Y 305.585,Z 453.037,A -85,B 0,C 180,E1 -15774.797,E2 -15774.797} C_VEL
LIN {X 0,Y 305.518,Z 453.047,A -85,B 0,C 180,E1 -15775.169,E2 -15775.169} C_VEL
LIN {X 0,Y 305.499,Z 453.049,A -85,B 0,C 180,E1 -15779.05,E2 -15779.05} C_VEL
LIN {X 0,Y 305.448,Z 453.05,A -85,B 0,C 180,E1 -15781.952,E2 -15781.952} C_VEL
LIN {X 0,Y 305.466,Z 453.061,A -85,B 0,C 180,E1 -15785.113,E2 -15785.113} C_VEL
LIN {X 0,Y 305.453,Z 453.046,A -85,B 0,C 180,E1 -15788.529,E2 -15788.529} C_VEL
LIN {X 0,Y 305.478,Z 453.05,A -85,B 0,C 180,E1 -15792.59,E2 -15792.59} C_VEL
LIN {X 0,Y 305.484,Z 453.049,A -85,B 0,C 180,E1 -15797.409,E2 -15797.409} C_VEL
LIN {X 0,Y 305.511,Z 453.055,A -85,B 0,C 180,E1 -15801.602,E2 -15801.602} C_VEL
LIN {X 0,Y 305.465,Z 453.048,A -85,B 0,C 180,E1 -15804.887,E2 -15804.887} C_VEL
LIN {X 0,Y 305.452,Z 453.056,A -85,B 0,C 180,E1 -15808.355,E2 -15808.355} C_VEL
LIN {X 0,Y 305.515,Z 453.04,A -85,B 0,C 180,E1 -15811.113,E2 -15811.113} C_VEL
LIN {X 0,Y 305.573,Z 453.044,A -85,B 0,C 180,E1 -15814.088,E2 -15814.088} C_VEL
LIN {X 0,Y 305.485,Z 453.053,A -85,B 0,C 180,E1 -15818.401,E2 -15818.401} C_VEL
LIN {X 0,Y 305.591,Z 453.042,A -85,B 0,C 180,E1 -15821.217,E2 -15821.217} C_VEL
LIN {X 0,Y 305.65,Z 453.029,A -85,B 0,C 180,E1 -15825.349,E2 -15825.349} C_VEL
LIN {X 0,Y 305.64,Z 453.023,A -85,B 0,C 180,E1 -15829.399,E2 -15829.399} C_VEL
LIN {X 0,Y 305.814,Z 453.009,A -85,B 0,C 180,E1 -15832.074,E2 -15832.074} C_VEL
LIN {X 0,Y 305.69,Z 453.028,A -85,B 0,C 180,E1 -15834.723,E2 -15834.723} C_VEL
LIN {X 0,Y 305.958,Z 452.991,A -85,B 0,C 180,E1 -15838.683,E2 -15838.683} C_VEL
LIN {X 0,Y 305.958,Z 452.999,A -85,B 0,C 180,E1 -15841.316,E2 -15841.316} C_VEL
LIN {X 0,Y 305.853,Z 453.005,A -85,B 0,C 180,E1 -15846.597,E2 -15846.597} C_VEL
LIN {X 0,Y 305.737,Z 453.026,A -85,B 0,C 180,E1 -15849.259,E2 -15849.259} C_VEL
LIN {X 0,Y 305.589,Z 453.03,A -85,B 0,C 180,E1 -15853.296,E2 -15853.296} C_VEL
LIN {X 0,Y 305.594,Z 453.042,A -85,B 0,C 180,E1 -15856.02,E2 -15856.02} C_VEL
LIN {X 0,Y 305.577,Z 453.03,A -85,B 0,C 180,E1 -15859.444,E2 -15859.444} C_VEL
LIN {X 0,Y 305.491,Z 453.053,A -85,B 0,C 180,E1 -15863.041,E2 -15863.041} C_VEL
LIN {X 0,Y 305.548,Z 453.049,A -85,B 0,C 180,E1 -15866.227,E2 -15866.227} C_VEL
LIN {X 0,Y 305.496,Z 453.053,A -85,B 0,C 180,E1 -15869.05,E2 -15869.05} C_VEL
LIN {X 0,Y 305.445,Z 453.064,A -85,B 0,C 180,E1 -15871.952,E2 -15871.952} C_VEL
LIN {X 0,Y 305.463,Z 453.06,A -85,B 0,C 180,E1 -15875.113,E2 -15875.113} C_VEL
LIN {X 0,Y 305.468,Z 453.058,A -85,B 0,C 180,E1 -15878.533,E2 -15878.533} C_VEL
LIN {X 0,Y 305.482,Z 453.056,A -85,B 0,C 180,E1 -15882.591,E2 -15882.591} C_VEL
LIN {X 0,Y 305.493,Z 453.055,A -85,B 0,C 180,E1 -15886.357,E2 -15886.357} C_VEL
LIN {X 0,Y 305.533,Z 453.18,A -85,B 0,C 180,E1 -15887.948,E2 -15887.948} C_VEL
LIN {X 0,Y 308.684,Z 464.178,A -85,B 0,C 180,E1 -15891.319,E2 -15891.319} C_VEL
LIN {X 0,Y 309.746,Z 467.999,A -85,B 0,C 180,E1 -15892.403,E2 -15892.403} C_VEL
LIN {X 0,Y 319.89,Z 488.862,A -85,B 0,C 180,E1 -15894.244,E2 -15894.244} C_VEL
LIN {X 0,Y 327.534,Z 506.273,A -85,B 0,C 180,E1 -15895.582,E2 -15895.582} C_VEL
LIN {X 0,Y 329.981,Z 520.98,A -85,B 0,C 180,E1 -15896.232,E2 -15896.232} C_VEL
LIN {X 0,Y 325.909,Z 635.2,A -85,B 0,C 180,E1 -15898.787,E2 -15898.787} C_VEL
LIN {X 0,Y 324.604,Z 650.99,A -85,B 0,C 180,E1 -15899.371,E2 -15899.371} C_VEL
LIN {X 0,Y 323.014,Z 665.567,A -85,B 0,C 180,E1 -15900.152,E2 -15900.152} C_VEL
LIN {X 0,Y 321.041,Z 680.305,A -85,B 0,C 180,E1 -15901.209,E2 -15901.209} C_VEL
LIN {X 0,Y 318.934,Z 693.709,A -85,B 0,C 180,E1 -15902.435,E2 -15902.435} C_VEL
LIN {X 0,Y 316.447,Z 707.337,A -85,B 0,C 180,E1 -15903.983,E2 -15903.983} C_VEL
LIN {X 0,Y 313.896,Z 719.713,A -85,B 0,C 180,E1 -15905.706,E2 -15905.706} C_VEL
LIN {X 0,Y 311.613,Z 730.976,A -85,B 0,C 180,E1 -15907.622,E2 -15907.622} C_VEL
LIN {X 0,Y 309.614,Z 741.264,A -85,B 0,C 180,E1 -15909.747,E2 -15909.747} C_VEL
LIN {X 0,Y 307.63,Z 750.471,A -85,B 0,C 180,E1 -15912.036,E2 -15912.036} C_VEL
LIN {X 0,Y 306.119,Z 758.288,A -85,B 0,C 180,E1 -15914.407,E2 -15914.407} C_VEL
LIN {X 0,Y 305.049,Z 764.432,A -85,B 0,C 180,E1 -15916.679,E2 -15916.679} C_VEL
LIN {X 0,Y 304.187,Z 770.223,A -85,B 0,C 180,E1 -15919.348,E2 -15919.348} C_VEL
LIN {X 0,Y 303.781,Z 774.636,A -85,B 0,C 180,E1 -15922.02,E2 -15922.02} C_VEL
LIN {X 0,Y 303.596,Z 777.768,A -85,B 0,C 180,E1 -15924.686,E2 -15924.686} C_VEL
LIN {X 0,Y 303.59,Z 779.68,A -85,B 0,C 180,E1 -15927.346,E2 -15927.346} C_VEL
LIN {X 0,Y 303.603,Z 780.368,A -85,B 0,C 180,E1 -15929.999,E2 -15929.999} C_VEL
LIN {X 0,Y 303.592,Z 779.903,A -85,B 0,C 180,E1 -15932.653,E2 -15932.653} C_VEL
LIN {X 0,Y 303.623,Z 778.085,A -85,B 0,C 180,E1 -15935.544,E2 -15935.544} C_VEL
LIN {X 0,Y 303.779,Z 775.496,A -85,B 0,C 180,E1 -15937.978,E2 -15937.978} C_VEL
LIN {X 0,Y 304.226,Z 771.467,A -85,B 0,C 180,E1 -15940.649,E2 -15940.649} C_VEL
LIN {X 0,Y 305.126,Z 766.078,A -85,B 0,C 180,E1 -15943.316,E2 -15943.316} C_VEL
LIN {X 0,Y 306.413,Z 759.231,A -85,B 0,C 180,E1 -15945.975,E2 -15945.975} C_VEL
LIN {X 0,Y 308.286,Z 750.748,A -85,B 0,C 180,E1 -15948.611,E2 -15948.611} C_VEL
LIN {X 0,Y 310.481,Z 741.711,A -85,B 0,C 180,E1 -15950.885,E2 -15950.885} C_VEL
LIN {X 0,Y 312.873,Z 731.218,A -85,B 0,C 180,E1 -15953.076,E2 -15953.076} C_VEL
LIN {X 0,Y 315.453,Z 719.772,A -85,B 0,C 180,E1 -15955.042,E2 -15955.042} C_VEL
LIN {X 0,Y 318.144,Z 707.626,A -85,B 0,C 180,E1 -15956.749,E2 -15956.749} C_VEL
LIN {X 0,Y 320.783,Z 694.319,A -85,B 0,C 180,E1 -15958.279,E2 -15958.279} C_VEL
LIN {X 0,Y 323.21,Z 680.357,A -85,B 0,C 180,E1 -15959.568,E2 -15959.568} C_VEL
LIN {X 0,Y 325.306,Z 666.124,A -85,B 0,C 180,E1 -15960.599,E2 -15960.599} C_VEL
LIN {X 0,Y 327.052,Z 652.151,A -85,B 0,C 180,E1 -15961.36,E2 -15961.36} C_VEL
LIN {X 0,Y 328.444,Z 637.445,A -85,B 0,C 180,E1 -15961.932,E2 -15961.932} C_VEL
LIN {X 0,Y 329.396,Z 616.646,A -85,B 0,C 180,E1 -15962.46,E2 -15962.46} C_VEL
LIN {X 0,Y 332.492,Z 537.18,A -85,B 0,C 180,E1 -15964.226,E2 -15964.226} C_VEL
LIN {X 0,Y 333.084,Z 521.006,A -85,B 0,C 180,E1 -15964.592,E2 -15964.592} C_VEL
LIN {X 0,Y 331.147,Z 509.103,A -85,B 0,C 180,E1 -15965.173,E2 -15965.173} C_VEL
LIN {X 0,Y 325.194,Z 495.829,A -85,B 0,C 180,E1 -15966.363,E2 -15966.363} C_VEL
LIN {X 0,Y 318.895,Z 483.096,A -85,B 0,C 180,E1 -15967.666,E2 -15967.666} C_VEL
LIN {X 0,Y 314.048,Z 474.36,A -85,B 0,C 180,E1 -15968.698,E2 -15968.698} C_VEL
LIN {X 0,Y 311.341,Z 469.686,A -85,B 0,C 180,E1 -15969.29,E2 -15969.29} C_VEL
LIN {X 0,Y 309.692,Z 466.512,A -85,B 0,C 180,E1 -15969.691,E2 -15969.691} C_VEL
LIN {X 0,Y 306.352,Z 455.68,A -85,B 0,C 180,E1 -15973.488,E2 -15973.488} C_VEL
LIN {X 0,Y 305.463,Z 453.064,A -85,B 0,C 180,E1 -15974.501,E2 -15974.501} C_VEL
LIN {X 0,Y 305.46,Z 453.061,A -85,B 0,C 180,E1 -15978.147,E2 -15978.147} C_VEL
LIN {X 0,Y 305.47,Z 453.058,A -85,B 0,C 180,E1 -15981.597,E2 -15981.597} C_VEL
LIN {X 0,Y 305.456,Z 453.058,A -85,B 0,C 180,E1 -15984.886,E2 -15984.886} C_VEL
LIN {X 0,Y 305.444,Z 453.064,A -85,B 0,C 180,E1 -15988.355,E2 -15988.355} C_VEL
LIN {X 0,Y 305.506,Z 453.055,A -85,B 0,C 180,E1 -15991.113,E2 -15991.113} C_VEL
LIN {X 0,Y 305.564,Z 453.046,A -85,B 0,C 180,E1 -15994.088,E2 -15994.088} C_VEL
LIN {X 0,Y 305.494,Z 453.055,A -85,B 0,C 180,E1 -15998.403,E2 -15998.403} C_VEL
LIN {X 0,Y 305.583,Z 453.045,A -85,B 0,C 180,E1 -16001.218,E2 -16001.218} C_VEL
LIN {X 0,Y 305.642,Z 453.037,A -85,B 0,C 180,E1 -16005.349,E2 -16005.349} C_VEL
LIN {X 0,Y 305.634,Z 453.037,A -85,B 0,C 180,E1 -16009.4,E2 -16009.4} C_VEL
